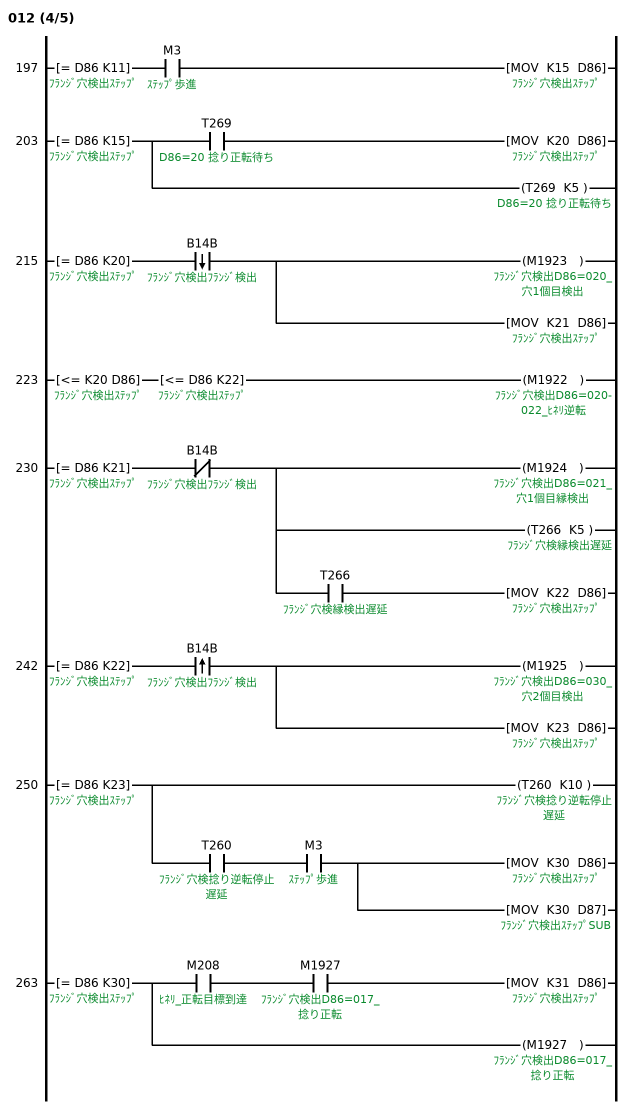
197   LD=     D86 K11  ; ﾌﾗﾝｼﾞ穴検出ｽﾃｯﾌﾟ
      AND     M3  ; ｽﾃｯﾌﾟ歩進
      MOV     K15 D86
203   LD=     D86 K15  ; ﾌﾗﾝｼﾞ穴検出ｽﾃｯﾌﾟ
      MPS
      AND     T269  ; D86=20 捻り正転待ち
      MOV     K20 D86
      MPP
      OUT     T269 K5  ; D86=20 捻り正転待ち
215   LD=     D86 K20  ; ﾌﾗﾝｼﾞ穴検出ｽﾃｯﾌﾟ
      ANDF    B14B  ; ﾌﾗﾝｼﾞ穴検出ﾌﾗﾝｼﾞ検出
      OUT     M1923  ; ﾌﾗﾝｼﾞ穴検出D86=020_穴1個目検出
      MOV     K21 D86
223   LD<=    K20 D86  ; ﾌﾗﾝｼﾞ穴検出ｽﾃｯﾌﾟ
      AND<=   D86 K22  ; ﾌﾗﾝｼﾞ穴検出ｽﾃｯﾌﾟ
      OUT     M1922  ; ﾌﾗﾝｼﾞ穴検出D86=020-022_ﾋﾈﾘ逆転
230   LD=     D86 K21  ; ﾌﾗﾝｼﾞ穴検出ｽﾃｯﾌﾟ
      ANI     B14B  ; ﾌﾗﾝｼﾞ穴検出ﾌﾗﾝｼﾞ検出
      OUT     M1924  ; ﾌﾗﾝｼﾞ穴検出D86=021_穴1個目縁検出
      OUT     T266 K5  ; ﾌﾗﾝｼﾞ穴検縁検出遅延
      AND     T266  ; ﾌﾗﾝｼﾞ穴検縁検出遅延
      MOV     K22 D86
242   LD=     D86 K22  ; ﾌﾗﾝｼﾞ穴検出ｽﾃｯﾌﾟ
      ANDP    B14B  ; ﾌﾗﾝｼﾞ穴検出ﾌﾗﾝｼﾞ検出
      OUT     M1925  ; ﾌﾗﾝｼﾞ穴検出D86=030_穴2個目検出
      MOV     K23 D86
250   LD=     D86 K23  ; ﾌﾗﾝｼﾞ穴検出ｽﾃｯﾌﾟ
      OUT     T260 K10  ; ﾌﾗﾝｼﾞ穴検捻り逆転停止遅延
      AND     T260  ; ﾌﾗﾝｼﾞ穴検捻り逆転停止遅延
      AND     M3  ; ｽﾃｯﾌﾟ歩進
      MOV     K30 D86
      MOV     K30 D87
263   LD=     D86 K30  ; ﾌﾗﾝｼﾞ穴検出ｽﾃｯﾌﾟ
      MPS
      AND     M208  ; ﾋﾈﾘ_正転目標到達
      AND     M1927  ; ﾌﾗﾝｼﾞ穴検出D86=017_捻り正転
      MOV     K31 D86
      MPP
      OUT     M1927  ; ﾌﾗﾝｼﾞ穴検出D86=017_捻り正転
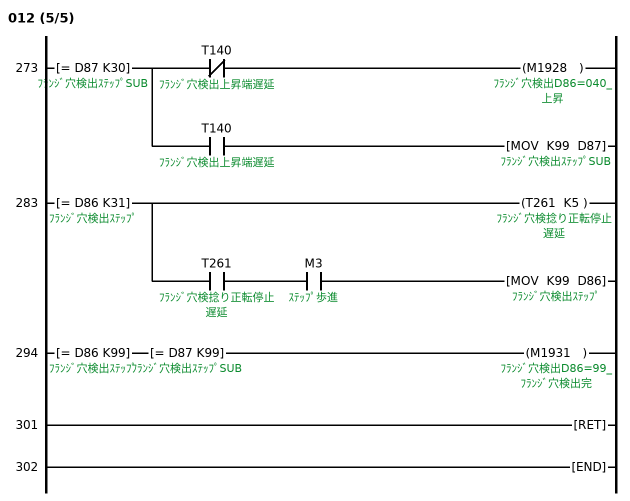
273   LD=     D87 K30  ; ﾌﾗﾝｼﾞ穴検出ｽﾃｯﾌﾟSUB
      MPS
      ANI     T140  ; ﾌﾗﾝｼﾞ穴検出上昇端遅延
      OUT     M1928  ; ﾌﾗﾝｼﾞ穴検出D86=040_上昇
      MPP
      AND     T140  ; ﾌﾗﾝｼﾞ穴検出上昇端遅延
      MOV     K99 D87
283   LD=     D86 K31  ; ﾌﾗﾝｼﾞ穴検出ｽﾃｯﾌﾟ
      OUT     T261 K5  ; ﾌﾗﾝｼﾞ穴検捻り正転停止遅延
      AND     T261  ; ﾌﾗﾝｼﾞ穴検捻り正転停止遅延
      AND     M3  ; ｽﾃｯﾌﾟ歩進
      MOV     K99 D86
294   LD=     D86 K99  ; ﾌﾗﾝｼﾞ穴検出ｽﾃｯﾌﾟ
      AND=    D87 K99  ; ﾌﾗﾝｼﾞ穴検出ｽﾃｯﾌﾟSUB
      OUT     M1931  ; ﾌﾗﾝｼﾞ穴検出D86=99_ﾌﾗﾝｼﾞ穴検出完
301   RET
302   END
END_PROGRAM

PROGRAM 013  // ひねり
; 
      P1300
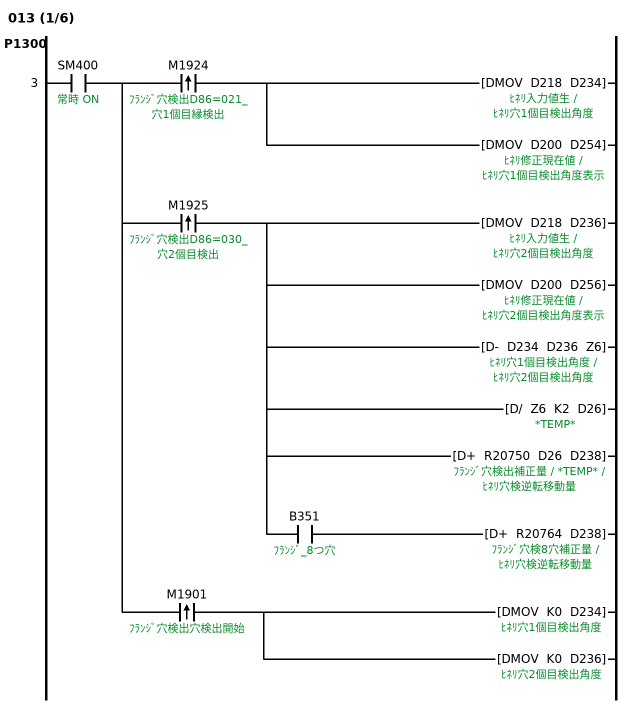
3     LD      SM400  ; 常時 ON
      MPS
      ANDP    M1924  ; ﾌﾗﾝｼﾞ穴検出D86=021_穴1個目縁検出
      DMOV    D218 D234  ; ﾋﾈﾘ入力値生 / ﾋﾈﾘ穴1個目検出角度
      DMOV    D200 D254  ; ﾋﾈﾘ修正現在値 / ﾋﾈﾘ穴1個目検出角度表示
      MRD
      ANDP    M1925  ; ﾌﾗﾝｼﾞ穴検出D86=030_穴2個目検出
      DMOV    D218 D236  ; ﾋﾈﾘ穴2個目検出角度
      DMOV    D200 D256  ; ﾋﾈﾘ穴2個目検出角度表示
      D-      D234 D236 Z6
      D/      Z6 K2 D26  ; *TEMP*
      D+      R20750 D26 D238  ; ﾌﾗﾝｼﾞ穴検出補正量 / ﾋﾈﾘ穴検逆転移動量
      AND     B351  ; ﾌﾗﾝｼﾞ_8つ穴
      D+      R20764 D238  ; ﾌﾗﾝｼﾞ穴検8穴補正量
      MPP
      ANDP    M1901  ; ﾌﾗﾝｼﾞ穴検出穴検出開始
      DMOV    K0 D234
      DMOV    K0 D236
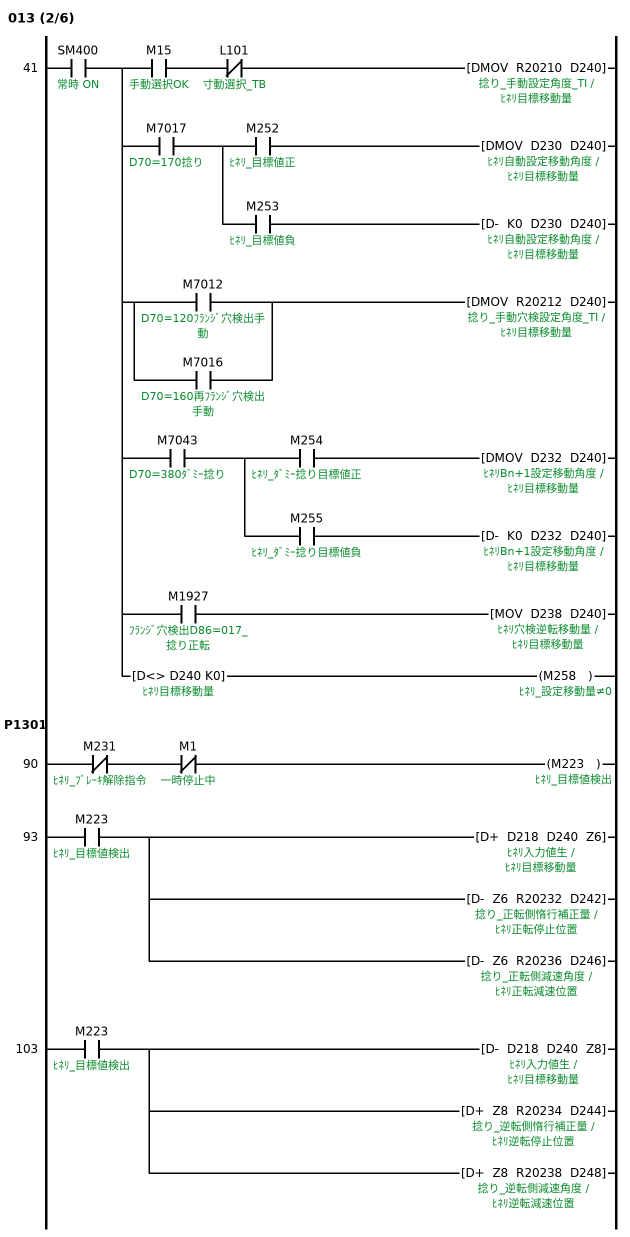
41    LD      SM400  ; 常時 ON
      MPS
      AND     M15  ; 手動選択OK
      ANI     L101  ; 寸動選択_TB
      DMOV    R20210 D240  ; 捻り_手動設定角度_TI / ﾋﾈﾘ目標移動量
      MRD
      AND     M7017  ; D70=170捻り
      MPS
      AND     M252  ; ﾋﾈﾘ_目標値正
      DMOV    D230 D240  ; ﾋﾈﾘ自動設定移動角度
      MPP
      AND     M253  ; ﾋﾈﾘ_目標値負
      D-      K0 D230 D240
      MRD
      LD      M7012  ; D70=120ﾌﾗﾝｼﾞ穴検出手動
      OR      M7016  ; D70=160再ﾌﾗﾝｼﾞ穴検出手動
      ANB
      DMOV    R20212 D240  ; 捻り_手動穴検設定角度_TI
      MRD
      AND     M7043  ; D70=380ﾀﾞﾐｰ捻り
      MPS
      AND     M254  ; ﾋﾈﾘ_ﾀﾞﾐｰ捻り目標値正
      DMOV    D232 D240  ; ﾋﾈﾘBn+1設定移動角度
      MPP
      AND     M255  ; ﾋﾈﾘ_ﾀﾞﾐｰ捻り目標値負
      D-      K0 D232 D240
      MRD
      AND     M1927  ; ﾌﾗﾝｼﾞ穴検出D86=017_捻り正転
      MOV     D238 D240
      MPP
      ANDD<>  D240 K0  ; ﾋﾈﾘ目標移動量
      OUT     M258  ; ﾋﾈﾘ_設定移動量≠0
; 
      P1301
90    LDI     M231  ; ﾋﾈﾘ_ﾌﾞﾚｰｷ解除指令
      ANI     M1  ; 一時停止中
      OUT     M223  ; ﾋﾈﾘ_目標値検出
93    LD      M223  ; ﾋﾈﾘ_目標値検出
      D+      D218 D240 Z6
      D-      Z6 R20232 D242  ; 捻り_正転側惰行補正量 / ﾋﾈﾘ正転停止位置
      D-      Z6 R20236 D246  ; 捻り_正転側減速角度 / ﾋﾈﾘ正転減速位置
103   LD      M223  ; ﾋﾈﾘ_目標値検出
      D-      D218 D240 Z8
      D+      Z8 R20234 D244  ; 捻り_逆転側惰行補正量 / ﾋﾈﾘ逆転停止位置
      D+      Z8 R20238 D248  ; 捻り_逆転側減速角度 / ﾋﾈﾘ逆転減速位置
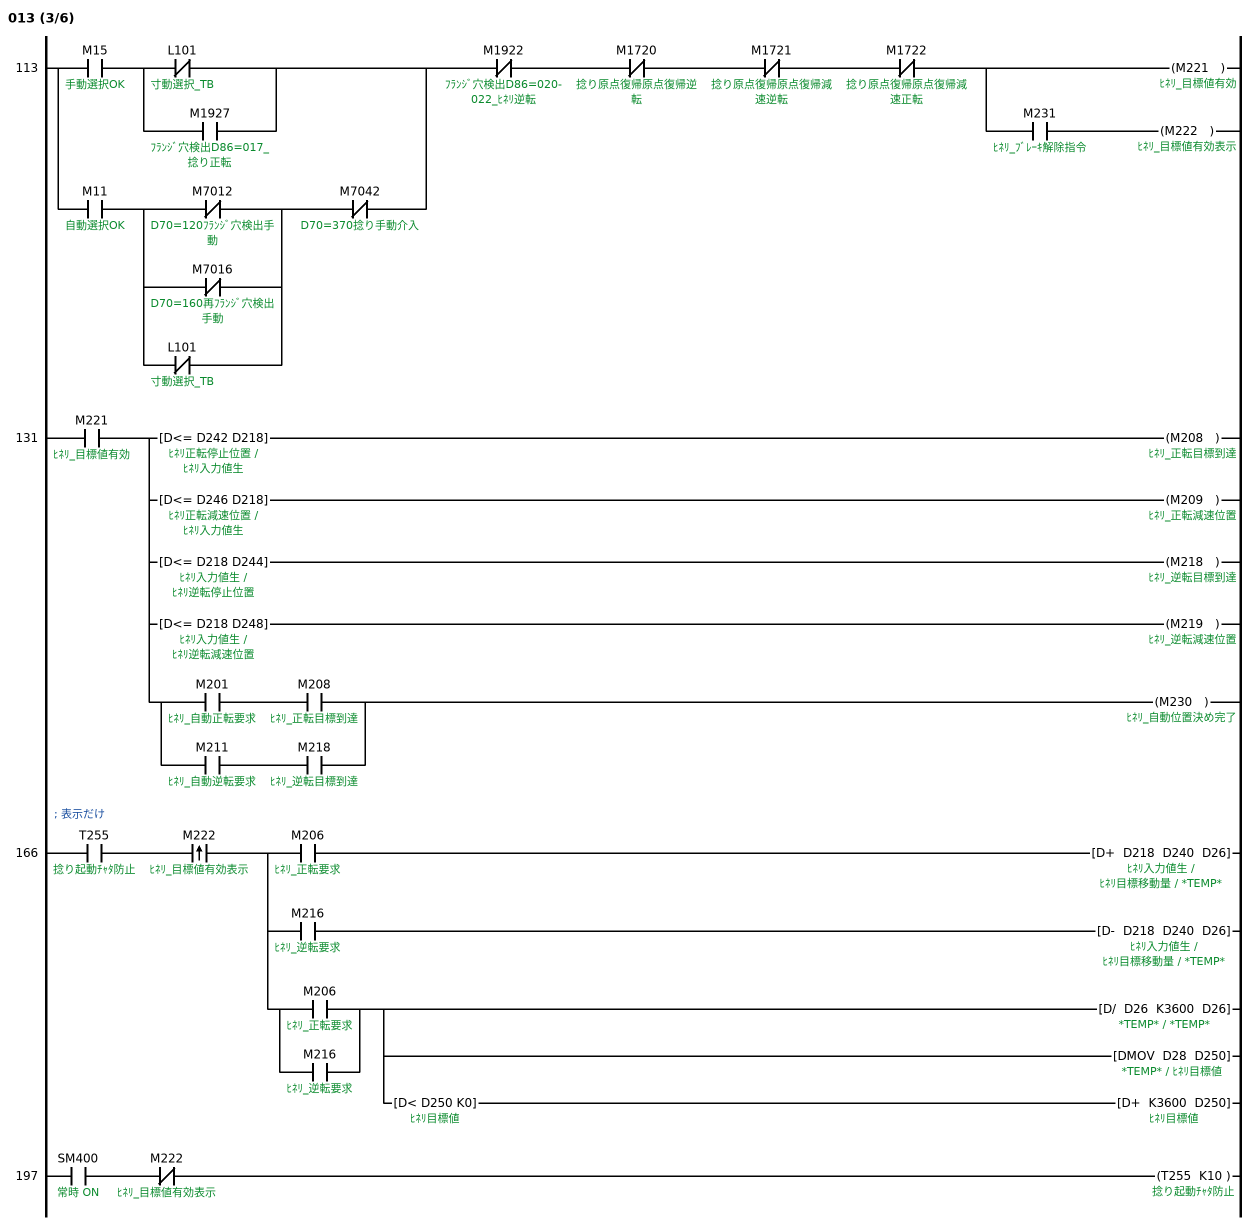
113   LD      M15  ; 手動選択OK
      LDI     L101  ; 寸動選択_TB
      OR      M1927  ; ﾌﾗﾝｼﾞ穴検出D86=017_捻り正転
      ANB
      LD      M11  ; 自動選択OK
      LDI     M7012  ; D70=120ﾌﾗﾝｼﾞ穴検出手動
      ORI     M7016  ; D70=160再ﾌﾗﾝｼﾞ穴検出手動
      ORI     L101  ; 寸動選択_TB
      ANB
      ANI     M7042  ; D70=370捻り手動介入
      ORB
      ANI     M1922  ; ﾌﾗﾝｼﾞ穴検出D86=020-022_ﾋﾈﾘ逆転
      ANI     M1720  ; 捻り原点復帰原点復帰逆転
      ANI     M1721  ; 捻り原点復帰原点復帰減速逆転
      ANI     M1722  ; 捻り原点復帰原点復帰減速正転
      OUT     M221  ; ﾋﾈﾘ_目標値有効
      AND     M231  ; ﾋﾈﾘ_ﾌﾞﾚｰｷ解除指令
      OUT     M222  ; ﾋﾈﾘ_目標値有効表示
131   LD      M221  ; ﾋﾈﾘ_目標値有効
      MPS
      ANDD<=  D242 D218  ; ﾋﾈﾘ正転停止位置 / ﾋﾈﾘ入力値生
      OUT     M208  ; ﾋﾈﾘ_正転目標到達
      MRD
      ANDD<=  D246 D218  ; ﾋﾈﾘ正転減速位置 / ﾋﾈﾘ入力値生
      OUT     M209  ; ﾋﾈﾘ_正転減速位置
      MRD
      ANDD<=  D218 D244  ; ﾋﾈﾘ入力値生 / ﾋﾈﾘ逆転停止位置
      OUT     M218  ; ﾋﾈﾘ_逆転目標到達
      MRD
      ANDD<=  D218 D248  ; ﾋﾈﾘ入力値生 / ﾋﾈﾘ逆転減速位置
      OUT     M219  ; ﾋﾈﾘ_逆転減速位置
      MPP
      LD      M201  ; ﾋﾈﾘ_自動正転要求
      AND     M208  ; ﾋﾈﾘ_正転目標到達
      LD      M211  ; ﾋﾈﾘ_自動逆転要求
      AND     M218  ; ﾋﾈﾘ_逆転目標到達
      ORB
      ANB
      OUT     M230  ; ﾋﾈﾘ_自動位置決め完了
; 表示だけ
166   LD      T255  ; 捻り起動ﾁｬﾀ防止
      ANDP    M222  ; ﾋﾈﾘ_目標値有効表示
      MPS
      AND     M206  ; ﾋﾈﾘ_正転要求
      D+      D218 D240 D26
      MRD
      AND     M216  ; ﾋﾈﾘ_逆転要求
      D-      D218 D240 D26
      MPP
      LD      M206  ; ﾋﾈﾘ_正転要求
      OR      M216  ; ﾋﾈﾘ_逆転要求
      ANB
      D/      D26 K3600 D26
      DMOV    D28 D250  ; *TEMP* / ﾋﾈﾘ目標値
      ANDD<   D250 K0  ; ﾋﾈﾘ目標値
      D+      K3600 D250
197   LD      SM400  ; 常時 ON
      ANI     M222  ; ﾋﾈﾘ_目標値有効表示
      OUT     T255 K10  ; 捻り起動ﾁｬﾀ防止
; 
      P1302
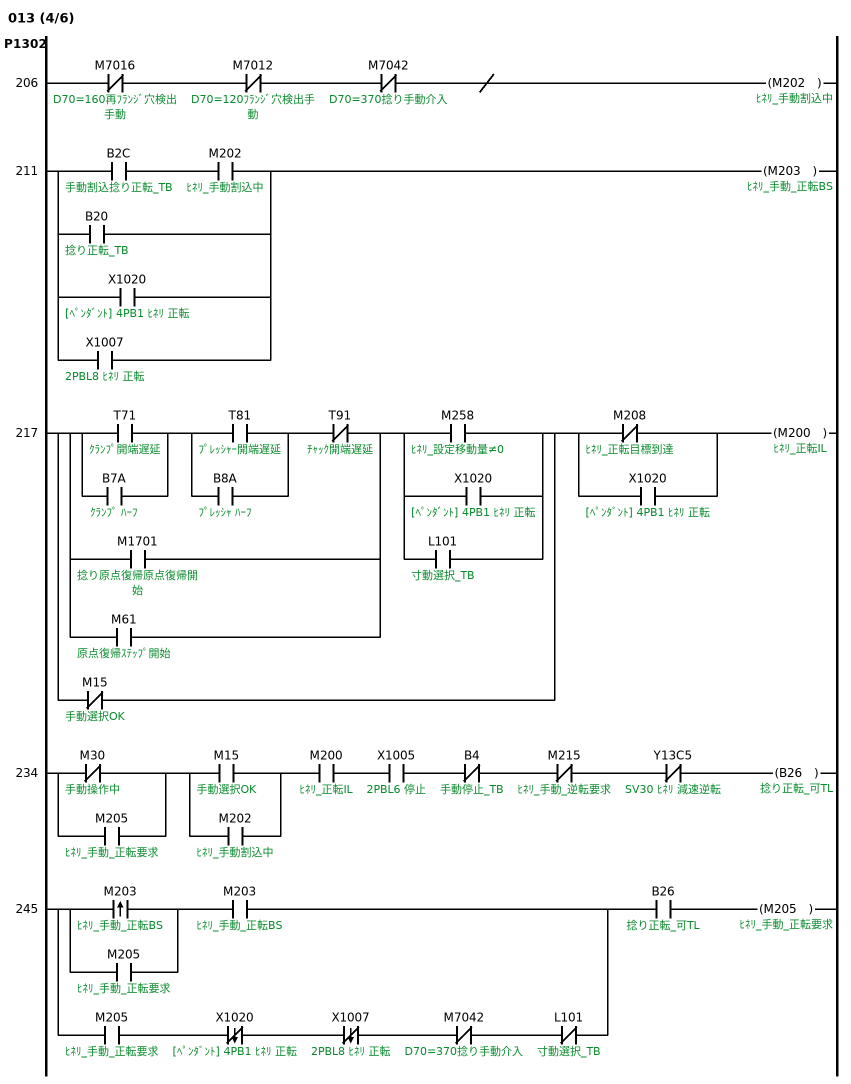
206   LDI     M7016  ; D70=160再ﾌﾗﾝｼﾞ穴検出手動
      ANI     M7012  ; D70=120ﾌﾗﾝｼﾞ穴検出手動
      ANI     M7042  ; D70=370捻り手動介入
      INV
      OUT     M202  ; ﾋﾈﾘ_手動割込中
211   LD      B2C  ; 手動割込捻り正転_TB
      AND     M202  ; ﾋﾈﾘ_手動割込中
      OR      B20  ; 捻り正転_TB
      OR      X1020  ; [ﾍﾟﾝﾀﾞﾝﾄ] 4PB1 ﾋﾈﾘ 正転
      OR      X1007  ; 2PBL8 ﾋﾈﾘ 正転
      OUT     M203  ; ﾋﾈﾘ_手動_正転BS
217   LD      T71  ; ｸﾗﾝﾌﾟ開端遅延
      OR      B7A  ; ｸﾗﾝﾌﾟ ﾊｰﾌ
      LD      T81  ; ﾌﾟﾚｯｼｬｰ開端遅延
      OR      B8A  ; ﾌﾟﾚｯｼｬ ﾊｰﾌ
      ANB
      ANI     T91  ; ﾁｬｯｸ開端遅延
      OR      M1701  ; 捻り原点復帰原点復帰開始
      OR      M61  ; 原点復帰ｽﾃｯﾌﾟ開始
      LD      M258  ; ﾋﾈﾘ_設定移動量≠0
      OR      X1020  ; [ﾍﾟﾝﾀﾞﾝﾄ] 4PB1 ﾋﾈﾘ 正転
      OR      L101  ; 寸動選択_TB
      ANB
      ORI     M15  ; 手動選択OK
      LDI     M208  ; ﾋﾈﾘ_正転目標到達
      OR      X1020  ; [ﾍﾟﾝﾀﾞﾝﾄ] 4PB1 ﾋﾈﾘ 正転
      ANB
      OUT     M200  ; ﾋﾈﾘ_正転IL
234   LDI     M30  ; 手動操作中
      OR      M205  ; ﾋﾈﾘ_手動_正転要求
      LD      M15  ; 手動選択OK
      OR      M202  ; ﾋﾈﾘ_手動割込中
      ANB
      AND     M200  ; ﾋﾈﾘ_正転IL
      AND     X1005  ; 2PBL6 停止
      ANI     B4  ; 手動停止_TB
      ANI     M215  ; ﾋﾈﾘ_手動_逆転要求
      ANI     Y13C5  ; SV30 ﾋﾈﾘ 減速逆転
      OUT     B26  ; 捻り正転_可TL
245   LDP     M203  ; ﾋﾈﾘ_手動_正転BS
      OR      M205  ; ﾋﾈﾘ_手動_正転要求
      AND     M203  ; ﾋﾈﾘ_手動_正転BS
      LD      M205  ; ﾋﾈﾘ_手動_正転要求
      ANDFI   X1020  ; [ﾍﾟﾝﾀﾞﾝﾄ] 4PB1 ﾋﾈﾘ 正転
      ANDFI   X1007  ; 2PBL8 ﾋﾈﾘ 正転
      ANI     M7042  ; D70=370捻り手動介入
      ANI     L101  ; 寸動選択_TB
      ORB
      AND     B26  ; 捻り正転_可TL
      OUT     M205  ; ﾋﾈﾘ_手動_正転要求
; 
      P1303
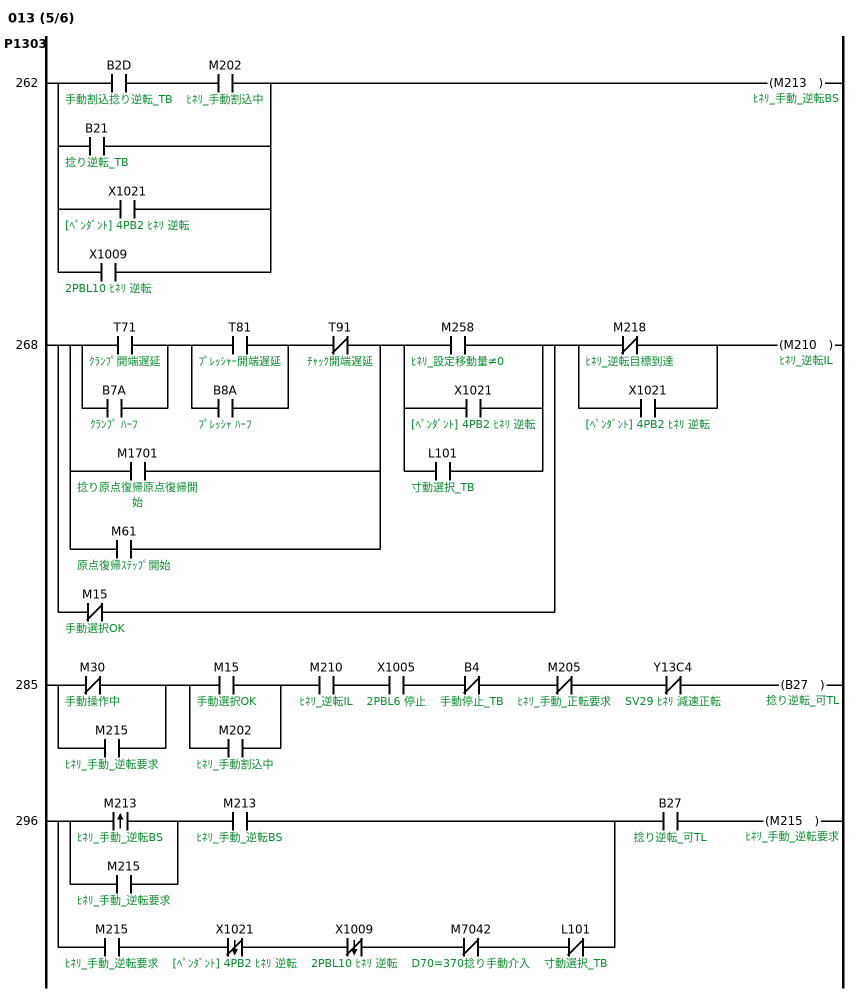
262   LD      B2D  ; 手動割込捻り逆転_TB
      AND     M202  ; ﾋﾈﾘ_手動割込中
      OR      B21  ; 捻り逆転_TB
      OR      X1021  ; [ﾍﾟﾝﾀﾞﾝﾄ] 4PB2 ﾋﾈﾘ 逆転
      OR      X1009  ; 2PBL10 ﾋﾈﾘ 逆転
      OUT     M213  ; ﾋﾈﾘ_手動_逆転BS
268   LD      T71  ; ｸﾗﾝﾌﾟ開端遅延
      OR      B7A  ; ｸﾗﾝﾌﾟ ﾊｰﾌ
      LD      T81  ; ﾌﾟﾚｯｼｬｰ開端遅延
      OR      B8A  ; ﾌﾟﾚｯｼｬ ﾊｰﾌ
      ANB
      ANI     T91  ; ﾁｬｯｸ開端遅延
      OR      M1701  ; 捻り原点復帰原点復帰開始
      OR      M61  ; 原点復帰ｽﾃｯﾌﾟ開始
      LD      M258  ; ﾋﾈﾘ_設定移動量≠0
      OR      X1021  ; [ﾍﾟﾝﾀﾞﾝﾄ] 4PB2 ﾋﾈﾘ 逆転
      OR      L101  ; 寸動選択_TB
      ANB
      ORI     M15  ; 手動選択OK
      LDI     M218  ; ﾋﾈﾘ_逆転目標到達
      OR      X1021  ; [ﾍﾟﾝﾀﾞﾝﾄ] 4PB2 ﾋﾈﾘ 逆転
      ANB
      OUT     M210  ; ﾋﾈﾘ_逆転IL
285   LDI     M30  ; 手動操作中
      OR      M215  ; ﾋﾈﾘ_手動_逆転要求
      LD      M15  ; 手動選択OK
      OR      M202  ; ﾋﾈﾘ_手動割込中
      ANB
      AND     M210  ; ﾋﾈﾘ_逆転IL
      AND     X1005  ; 2PBL6 停止
      ANI     B4  ; 手動停止_TB
      ANI     M205  ; ﾋﾈﾘ_手動_正転要求
      ANI     Y13C4  ; SV29 ﾋﾈﾘ 減速正転
      OUT     B27  ; 捻り逆転_可TL
296   LDP     M213  ; ﾋﾈﾘ_手動_逆転BS
      OR      M215  ; ﾋﾈﾘ_手動_逆転要求
      AND     M213  ; ﾋﾈﾘ_手動_逆転BS
      LD      M215  ; ﾋﾈﾘ_手動_逆転要求
      ANDFI   X1021  ; [ﾍﾟﾝﾀﾞﾝﾄ] 4PB2 ﾋﾈﾘ 逆転
      ANDFI   X1009  ; 2PBL10 ﾋﾈﾘ 逆転
      ANI     M7042  ; D70=370捻り手動介入
      ANI     L101  ; 寸動選択_TB
      ORB
      AND     B27  ; 捻り逆転_可TL
      OUT     M215  ; ﾋﾈﾘ_手動_逆転要求
; 
      P1306
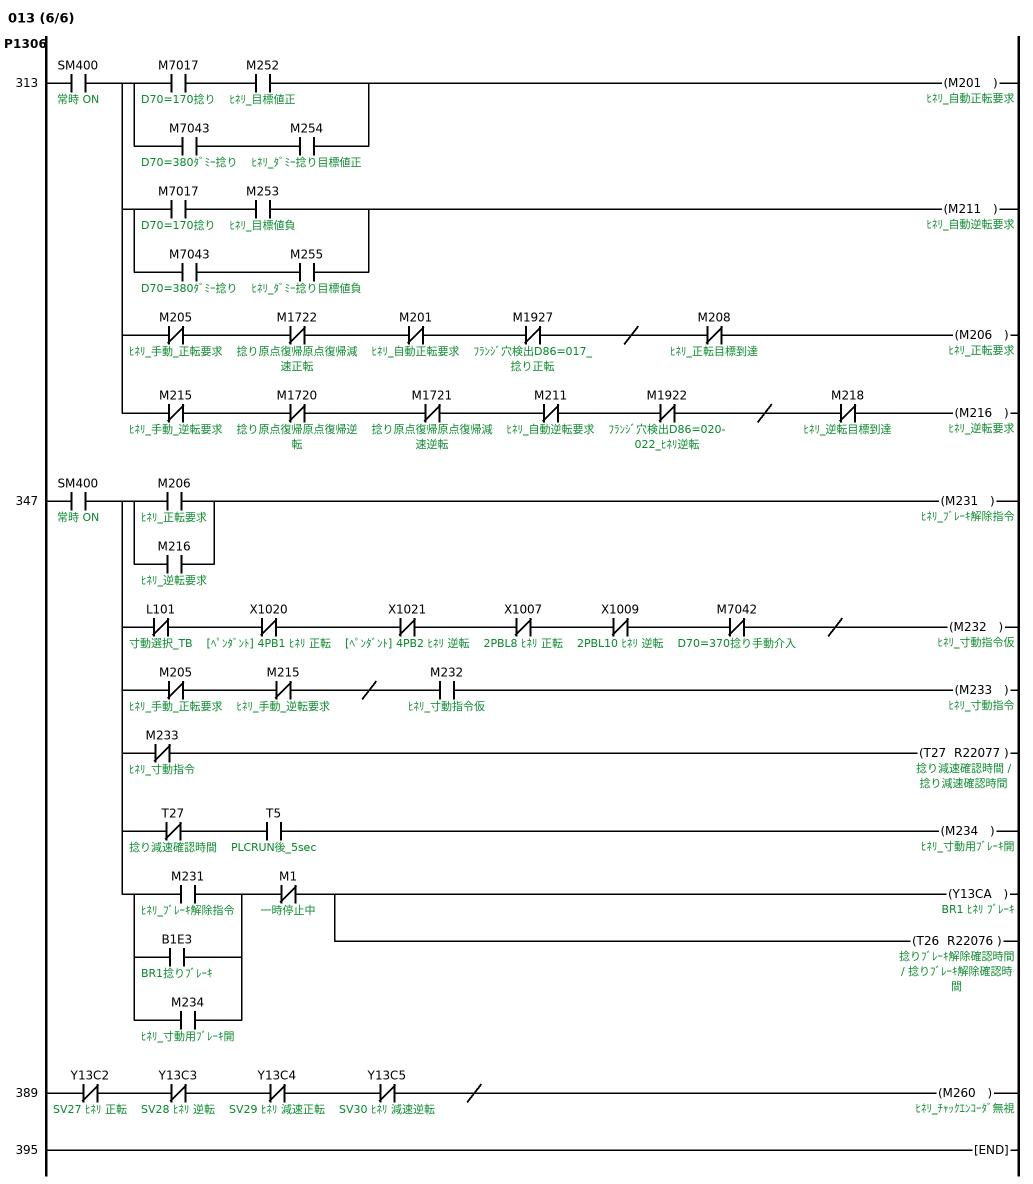
313   LD      SM400  ; 常時 ON
      MPS
      LD      M7017  ; D70=170捻り
      AND     M252  ; ﾋﾈﾘ_目標値正
      LD      M7043  ; D70=380ﾀﾞﾐｰ捻り
      AND     M254  ; ﾋﾈﾘ_ﾀﾞﾐｰ捻り目標値正
      ORB
      ANB
      OUT     M201  ; ﾋﾈﾘ_自動正転要求
      MRD
      LD      M7017  ; D70=170捻り
      AND     M253  ; ﾋﾈﾘ_目標値負
      LD      M7043  ; D70=380ﾀﾞﾐｰ捻り
      AND     M255  ; ﾋﾈﾘ_ﾀﾞﾐｰ捻り目標値負
      ORB
      ANB
      OUT     M211  ; ﾋﾈﾘ_自動逆転要求
      MRD
      ANI     M205  ; ﾋﾈﾘ_手動_正転要求
      ANI     M1722  ; 捻り原点復帰原点復帰減速正転
      ANI     M201  ; ﾋﾈﾘ_自動正転要求
      ANI     M1927  ; ﾌﾗﾝｼﾞ穴検出D86=017_捻り正転
      INV
      ANI     M208  ; ﾋﾈﾘ_正転目標到達
      OUT     M206  ; ﾋﾈﾘ_正転要求
      MPP
      ANI     M215  ; ﾋﾈﾘ_手動_逆転要求
      ANI     M1720  ; 捻り原点復帰原点復帰逆転
      ANI     M1721  ; 捻り原点復帰原点復帰減速逆転
      ANI     M211  ; ﾋﾈﾘ_自動逆転要求
      ANI     M1922  ; ﾌﾗﾝｼﾞ穴検出D86=020-022_ﾋﾈﾘ逆転
      INV
      ANI     M218  ; ﾋﾈﾘ_逆転目標到達
      OUT     M216  ; ﾋﾈﾘ_逆転要求
347   LD      SM400  ; 常時 ON
      MPS
      LD      M206  ; ﾋﾈﾘ_正転要求
      OR      M216  ; ﾋﾈﾘ_逆転要求
      ANB
      OUT     M231  ; ﾋﾈﾘ_ﾌﾞﾚｰｷ解除指令
      MRD
      ANI     L101  ; 寸動選択_TB
      ANI     X1020  ; [ﾍﾟﾝﾀﾞﾝﾄ] 4PB1 ﾋﾈﾘ 正転
      ANI     X1021  ; [ﾍﾟﾝﾀﾞﾝﾄ] 4PB2 ﾋﾈﾘ 逆転
      ANI     X1007  ; 2PBL8 ﾋﾈﾘ 正転
      ANI     X1009  ; 2PBL10 ﾋﾈﾘ 逆転
      ANI     M7042  ; D70=370捻り手動介入
      INV
      OUT     M232  ; ﾋﾈﾘ_寸動指令仮
      MRD
      ANI     M205  ; ﾋﾈﾘ_手動_正転要求
      ANI     M215  ; ﾋﾈﾘ_手動_逆転要求
      INV
      AND     M232  ; ﾋﾈﾘ_寸動指令仮
      OUT     M233  ; ﾋﾈﾘ_寸動指令
      MRD
      ANI     M233  ; ﾋﾈﾘ_寸動指令
      OUT     T27 R22077  ; 捻り減速確認時間 / 捻り減速確認時間
      MRD
      ANI     T27  ; 捻り減速確認時間
      AND     T5  ; PLCRUN後_5sec
      OUT     M234  ; ﾋﾈﾘ_寸動用ﾌﾞﾚｰｷ開
      MPP
      LD      M231  ; ﾋﾈﾘ_ﾌﾞﾚｰｷ解除指令
      OR      B1E3  ; BR1捻りﾌﾞﾚｰｷ
      OR      M234  ; ﾋﾈﾘ_寸動用ﾌﾞﾚｰｷ開
      ANB
      ANI     M1  ; 一時停止中
      OUT     Y13CA  ; BR1 ﾋﾈﾘ ﾌﾞﾚｰｷ
      OUT     T26 R22076  ; 捻りﾌﾞﾚｰｷ解除確認時間 / 捻りﾌﾞﾚｰｷ解除確認時間
389   LDI     Y13C2  ; SV27 ﾋﾈﾘ 正転
      ANI     Y13C3  ; SV28 ﾋﾈﾘ 逆転
      ANI     Y13C4  ; SV29 ﾋﾈﾘ 減速正転
      ANI     Y13C5  ; SV30 ﾋﾈﾘ 減速逆転
      INV
      OUT     M260  ; ﾋﾈﾘ_ﾁｬｯｸｴﾝｺｰﾀﾞ無視
395   END
END_PROGRAM

PROGRAM 018  // 送り
; 
      P1802
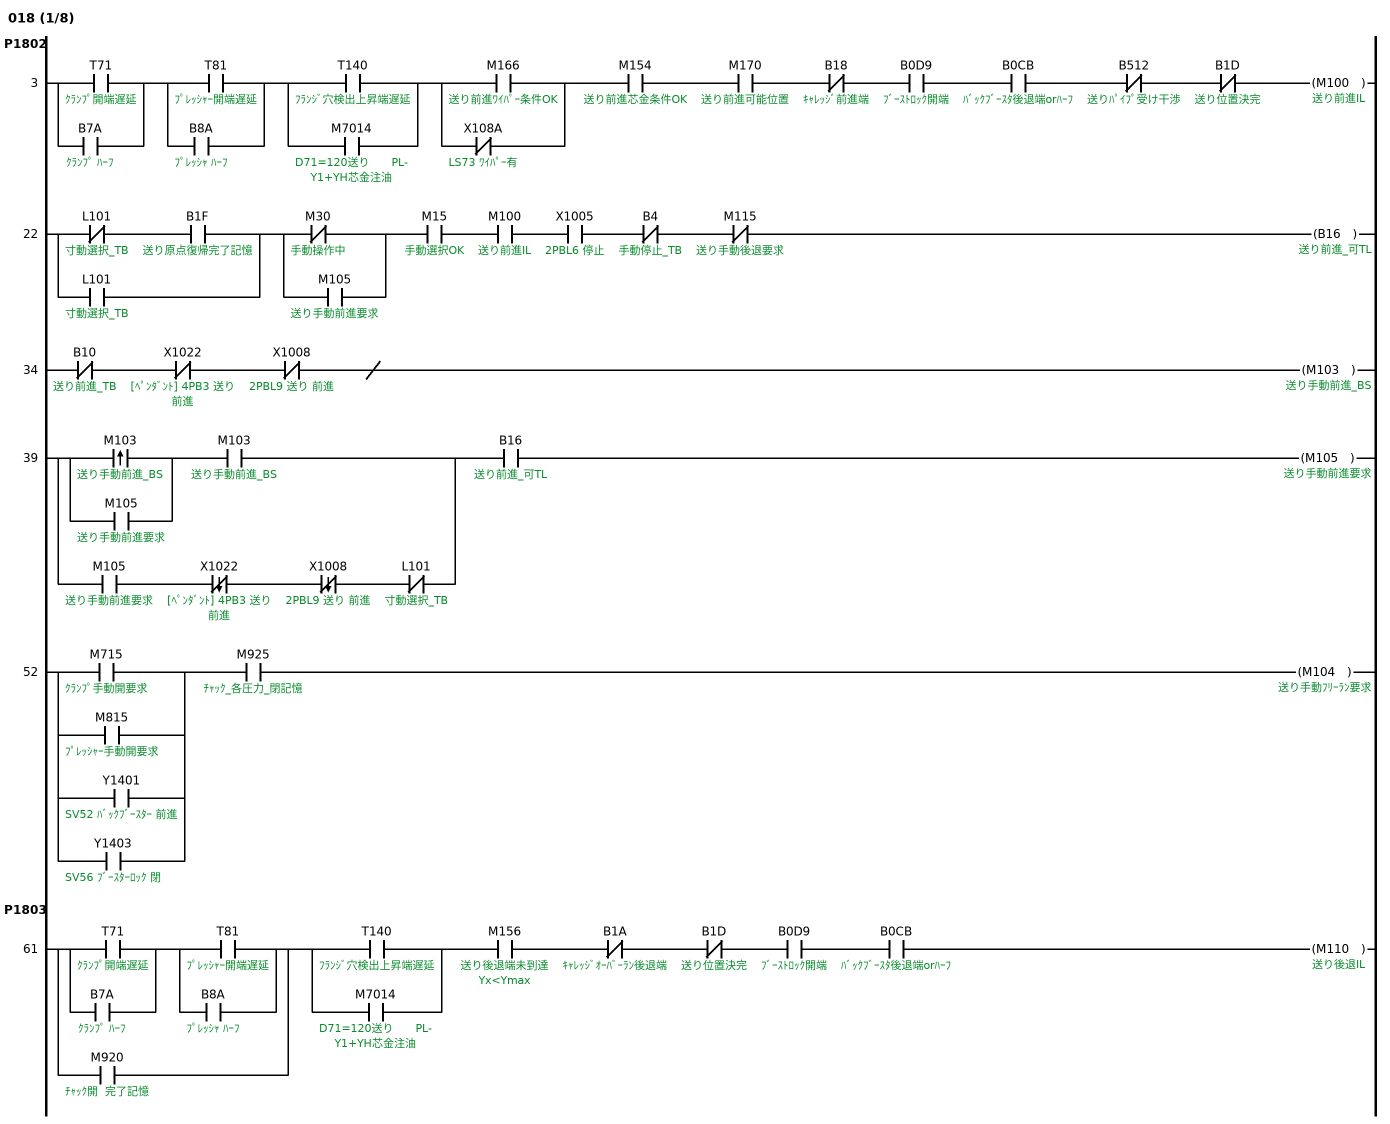
3     LD      T71  ; ｸﾗﾝﾌﾟ開端遅延
      OR      B7A  ; ｸﾗﾝﾌﾟ ﾊｰﾌ
      LD      T81  ; ﾌﾟﾚｯｼｬｰ開端遅延
      OR      B8A  ; ﾌﾟﾚｯｼｬ ﾊｰﾌ
      ANB
      LD      T140  ; ﾌﾗﾝｼﾞ穴検出上昇端遅延
      OR      M7014  ; D71=120送り　　PL-Y1+YH芯金注油
      ANB
      LD      M166  ; 送り前進ﾜｲﾊﾟｰ条件OK
      ORI     X108A  ; LS73 ﾜｲﾊﾟｰ有
      ANB
      AND     M154  ; 送り前進芯金条件OK
      AND     M170  ; 送り前進可能位置
      ANI     B18  ; ｷｬﾚｯｼﾞ前進端
      AND     B0D9  ; ﾌﾞｰｽﾄﾛｯｸ開端
      AND     B0CB  ; ﾊﾞｯｸﾌﾞｰｽﾀ後退端orﾊｰﾌ
      ANI     B512  ; 送りﾊﾟｲﾌﾟ受け干渉
      ANI     B1D  ; 送り位置決完
      OUT     M100  ; 送り前進IL
22    LDI     L101  ; 寸動選択_TB
      AND     B1F  ; 送り原点復帰完了記憶
      OR      L101  ; 寸動選択_TB
      LDI     M30  ; 手動操作中
      OR      M105  ; 送り手動前進要求
      ANB
      AND     M15  ; 手動選択OK
      AND     M100  ; 送り前進IL
      AND     X1005  ; 2PBL6 停止
      ANI     B4  ; 手動停止_TB
      ANI     M115  ; 送り手動後退要求
      OUT     B16  ; 送り前進_可TL
34    LDI     B10  ; 送り前進_TB
      ANI     X1022  ; [ﾍﾟﾝﾀﾞﾝﾄ] 4PB3 送り 前進
      ANI     X1008  ; 2PBL9 送り 前進
      INV
      OUT     M103  ; 送り手動前進_BS
39    LDP     M103  ; 送り手動前進_BS
      OR      M105  ; 送り手動前進要求
      AND     M103  ; 送り手動前進_BS
      LD      M105  ; 送り手動前進要求
      ANDFI   X1022  ; [ﾍﾟﾝﾀﾞﾝﾄ] 4PB3 送り 前進
      ANDFI   X1008  ; 2PBL9 送り 前進
      ANI     L101  ; 寸動選択_TB
      ORB
      AND     B16  ; 送り前進_可TL
      OUT     M105  ; 送り手動前進要求
52    LD      M715  ; ｸﾗﾝﾌﾟ手動開要求
      OR      M815  ; ﾌﾟﾚｯｼｬｰ手動開要求
      OR      Y1401  ; SV52 ﾊﾞｯｸﾌﾞｰｽﾀｰ 前進
      OR      Y1403  ; SV56 ﾌﾞｰｽﾀｰﾛｯｸ 閉
      AND     M925  ; ﾁｬｯｸ_各圧力_閉記憶
      OUT     M104  ; 送り手動ﾌﾘｰﾗﾝ要求
; 
      P1803
61    LD      T71  ; ｸﾗﾝﾌﾟ開端遅延
      OR      B7A  ; ｸﾗﾝﾌﾟ ﾊｰﾌ
      LD      T81  ; ﾌﾟﾚｯｼｬｰ開端遅延
      OR      B8A  ; ﾌﾟﾚｯｼｬ ﾊｰﾌ
      ANB
      OR      M920  ; ﾁｬｯｸ開  完了記憶
      LD      T140  ; ﾌﾗﾝｼﾞ穴検出上昇端遅延
      OR      M7014  ; D71=120送り　　PL-Y1+YH芯金注油
      ANB
      AND     M156  ; 送り後退端未到達 Yx<Ymax
      ANI     B1A  ; ｷｬﾚｯｼﾞｵｰﾊﾞｰﾗﾝ後退端
      ANI     B1D  ; 送り位置決完
      AND     B0D9  ; ﾌﾞｰｽﾄﾛｯｸ開端
      AND     B0CB  ; ﾊﾞｯｸﾌﾞｰｽﾀ後退端orﾊｰﾌ
      OUT     M110  ; 送り後退IL
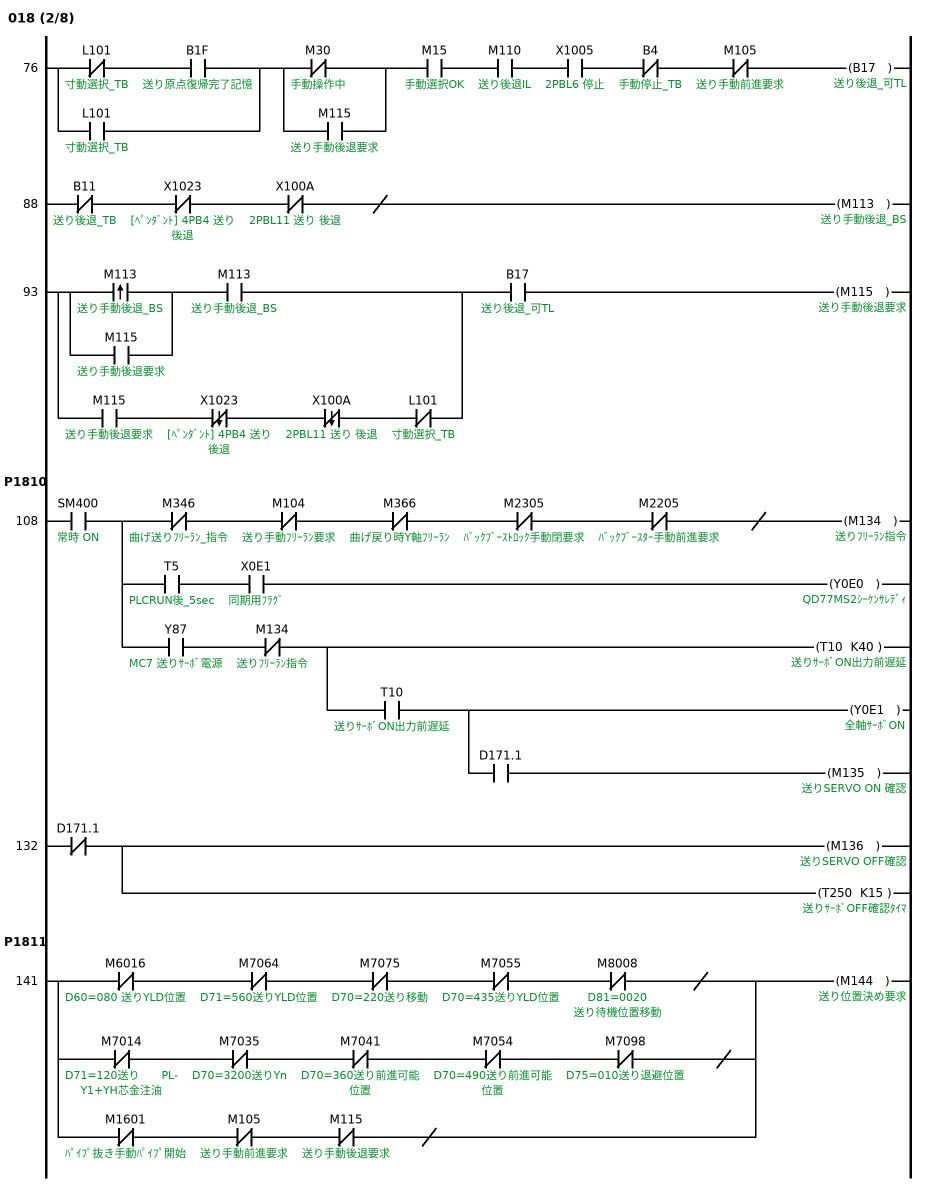
76    LDI     L101  ; 寸動選択_TB
      AND     B1F  ; 送り原点復帰完了記憶
      OR      L101  ; 寸動選択_TB
      LDI     M30  ; 手動操作中
      OR      M115  ; 送り手動後退要求
      ANB
      AND     M15  ; 手動選択OK
      AND     M110  ; 送り後退IL
      AND     X1005  ; 2PBL6 停止
      ANI     B4  ; 手動停止_TB
      ANI     M105  ; 送り手動前進要求
      OUT     B17  ; 送り後退_可TL
88    LDI     B11  ; 送り後退_TB
      ANI     X1023  ; [ﾍﾟﾝﾀﾞﾝﾄ] 4PB4 送り 後退
      ANI     X100A  ; 2PBL11 送り 後退
      INV
      OUT     M113  ; 送り手動後退_BS
93    LDP     M113  ; 送り手動後退_BS
      OR      M115  ; 送り手動後退要求
      AND     M113  ; 送り手動後退_BS
      LD      M115  ; 送り手動後退要求
      ANDFI   X1023  ; [ﾍﾟﾝﾀﾞﾝﾄ] 4PB4 送り 後退
      ANDFI   X100A  ; 2PBL11 送り 後退
      ANI     L101  ; 寸動選択_TB
      ORB
      AND     B17  ; 送り後退_可TL
      OUT     M115  ; 送り手動後退要求
; 
      P1810
108   LD      SM400  ; 常時 ON
      MPS
      ANI     M346  ; 曲げ送りﾌﾘｰﾗﾝ_指令
      ANI     M104  ; 送り手動ﾌﾘｰﾗﾝ要求
      ANI     M366  ; 曲げ戻り時Y軸ﾌﾘｰﾗﾝ
      ANI     M2305  ; ﾊﾞｯｸﾌﾞｰｽﾄﾛｯｸ手動閉要求
      ANI     M2205  ; ﾊﾞｯｸﾌﾞｰｽﾀｰ手動前進要求
      INV
      OUT     M134  ; 送りﾌﾘｰﾗﾝ指令
      MRD
      AND     T5  ; PLCRUN後_5sec
      AND     X0E1  ; 同期用ﾌﾗｸﾞ
      OUT     Y0E0  ; QD77MS2ｼｰｹﾝｻﾚﾃﾞｨ
      MPP
      AND     Y87  ; MC7 送りｻｰﾎﾞ電源
      ANI     M134  ; 送りﾌﾘｰﾗﾝ指令
      OUT     T10 K40  ; 送りｻｰﾎﾞON出力前遅延
      AND     T10  ; 送りｻｰﾎﾞON出力前遅延
      OUT     Y0E1  ; 全軸ｻｰﾎﾞON
      AND     D171.1
      OUT     M135  ; 送りSERVO ON 確認
132   LDI     D171.1
      OUT     M136  ; 送りSERVO OFF確認
      OUT     T250 K15  ; 送りｻｰﾎﾞOFF確認ﾀｲﾏ
; 
      P1811
141   LDI     M6016  ; D60=080 送りYLD位置
      ANI     M7064  ; D71=560送りYLD位置
      ANI     M7075  ; D70=220送り移動
      ANI     M7055  ; D70=435送りYLD位置
      ANI     M8008  ; D81=0020 送り待機位置移動
      INV
      LDI     M7014  ; D71=120送り　　PL-Y1+YH芯金注油
      ANI     M7035  ; D70=3200送りYn
      ANI     M7041  ; D70=360送り前進可能位置
      ANI     M7054  ; D70=490送り前進可能位置
      ANI     M7098  ; D75=010送り退避位置
      INV
      ORB
      LDI     M1601  ; ﾊﾟｲﾌﾟ抜き手動ﾊﾟｲﾌﾟ開始
      ANI     M105  ; 送り手動前進要求
      ANI     M115  ; 送り手動後退要求
      INV
      ORB
      OUT     M144  ; 送り位置決め要求
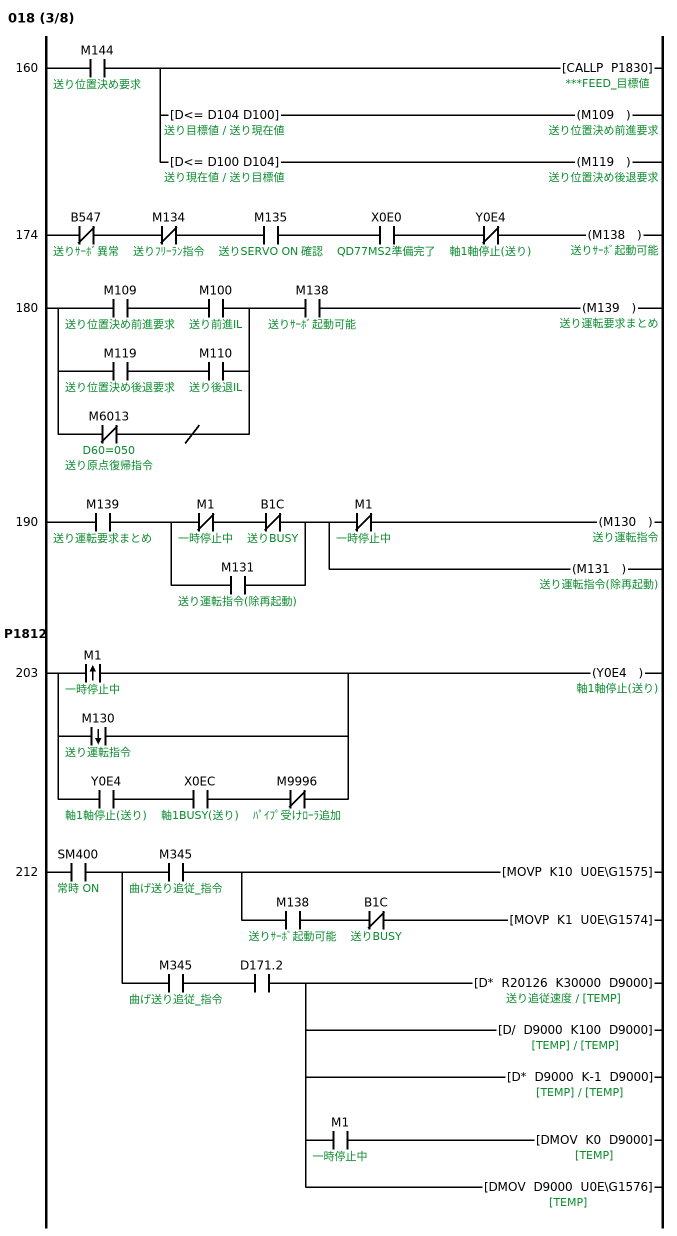
160   LD      M144  ; 送り位置決め要求
      CALLP   P1830  ; ***FEED_目標値
      MPS
      ANDD<=  D104 D100  ; 送り目標値 / 送り現在値
      OUT     M109  ; 送り位置決め前進要求
      MPP
      ANDD<=  D100 D104  ; 送り現在値 / 送り目標値
      OUT     M119  ; 送り位置決め後退要求
174   LDI     B547  ; 送りｻｰﾎﾞ異常
      ANI     M134  ; 送りﾌﾘｰﾗﾝ指令
      AND     M135  ; 送りSERVO ON 確認
      AND     X0E0  ; QD77MS2準備完了
      ANI     Y0E4  ; 軸1軸停止(送り)
      OUT     M138  ; 送りｻｰﾎﾞ起動可能
180   LD      M109  ; 送り位置決め前進要求
      AND     M100  ; 送り前進IL
      LD      M119  ; 送り位置決め後退要求
      AND     M110  ; 送り後退IL
      ORB
      LDI     M6013  ; D60=050 送り原点復帰指令
      INV
      ORB
      AND     M138  ; 送りｻｰﾎﾞ起動可能
      OUT     M139  ; 送り運転要求まとめ
190   LD      M139  ; 送り運転要求まとめ
      LDI     M1  ; 一時停止中
      ANI     B1C  ; 送りBUSY
      OR      M131  ; 送り運転指令(除再起動)
      ANB
      MPS
      ANI     M1  ; 一時停止中
      OUT     M130  ; 送り運転指令
      MPP
      OUT     M131  ; 送り運転指令(除再起動)
; 
      P1812
203   LDP     M1  ; 一時停止中
      ORF     M130  ; 送り運転指令
      LD      Y0E4  ; 軸1軸停止(送り)
      AND     X0EC  ; 軸1BUSY(送り)
      ANI     M9996  ; ﾊﾟｲﾌﾟ受けﾛｰﾗ追加
      ORB
      OUT     Y0E4  ; 軸1軸停止(送り)
212   LD      SM400  ; 常時 ON
      MPS
      AND     M345  ; 曲げ送り追従_指令
      MOVP    K10 U0E\G1575
      AND     M138  ; 送りｻｰﾎﾞ起動可能
      ANI     B1C  ; 送りBUSY
      MOVP    K1 U0E\G1574
      MPP
      AND     M345  ; 曲げ送り追従_指令
      AND     D171.2
      D*      R20126 K30000 D9000  ; 送り追従速度 / [TEMP]
      D/      D9000 K100 D9000
      D*      D9000 K-1 D9000
      MPS
      AND     M1  ; 一時停止中
      DMOV    K0 D9000
      MPP
      DMOV    D9000 U0E\G1576
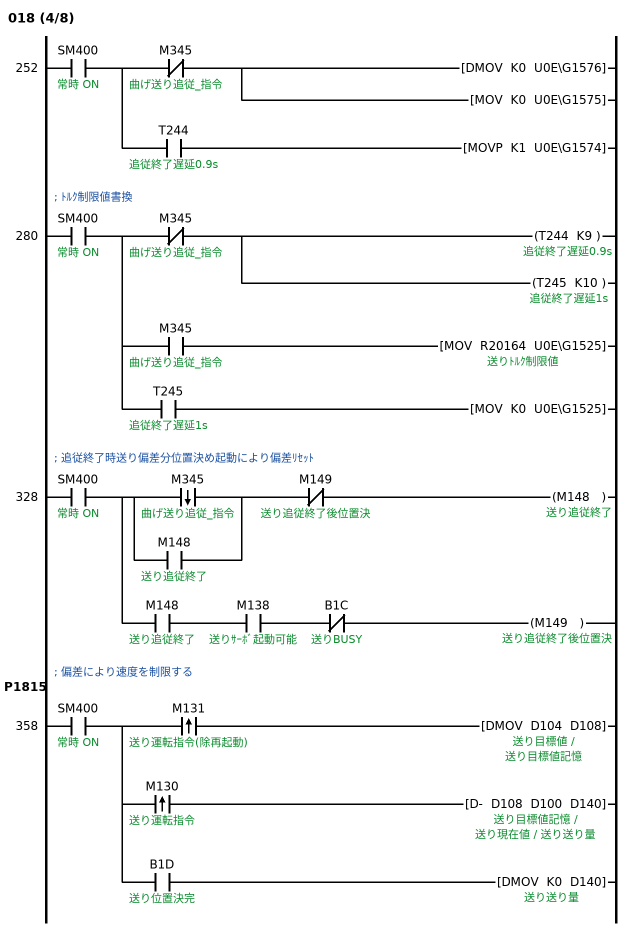
252   LD      SM400  ; 常時 ON
      MPS
      ANI     M345  ; 曲げ送り追従_指令
      DMOV    K0 U0E\G1576
      MOV     K0 U0E\G1575
      MPP
      AND     T244  ; 追従終了遅延0.9s
      MOVP    K1 U0E\G1574
; ﾄﾙｸ制限値書換
280   LD      SM400  ; 常時 ON
      MPS
      ANI     M345  ; 曲げ送り追従_指令
      OUT     T244 K9  ; 追従終了遅延0.9s
      OUT     T245 K10  ; 追従終了遅延1s
      MRD
      AND     M345  ; 曲げ送り追従_指令
      MOV     R20164 U0E\G1525  ; 送りﾄﾙｸ制限値
      MPP
      AND     T245  ; 追従終了遅延1s
      MOV     K0 U0E\G1525
; 追従終了時送り偏差分位置決め起動により偏差ﾘｾｯﾄ
328   LD      SM400  ; 常時 ON
      MPS
      LDF     M345  ; 曲げ送り追従_指令
      OR      M148  ; 送り追従終了
      ANB
      ANI     M149  ; 送り追従終了後位置決
      OUT     M148  ; 送り追従終了
      MPP
      AND     M148  ; 送り追従終了
      AND     M138  ; 送りｻｰﾎﾞ起動可能
      ANI     B1C  ; 送りBUSY
      OUT     M149  ; 送り追従終了後位置決
; 偏差により速度を制限する
; 
      P1815
358   LD      SM400  ; 常時 ON
      MPS
      ANDP    M131  ; 送り運転指令(除再起動)
      DMOV    D104 D108  ; 送り目標値記憶
      MRD
      ANDP    M130  ; 送り運転指令
      D-      D108 D100 D140  ; 送り送り量
      MPP
      AND     B1D  ; 送り位置決完
      DMOV    K0 D140
; 
      P1816
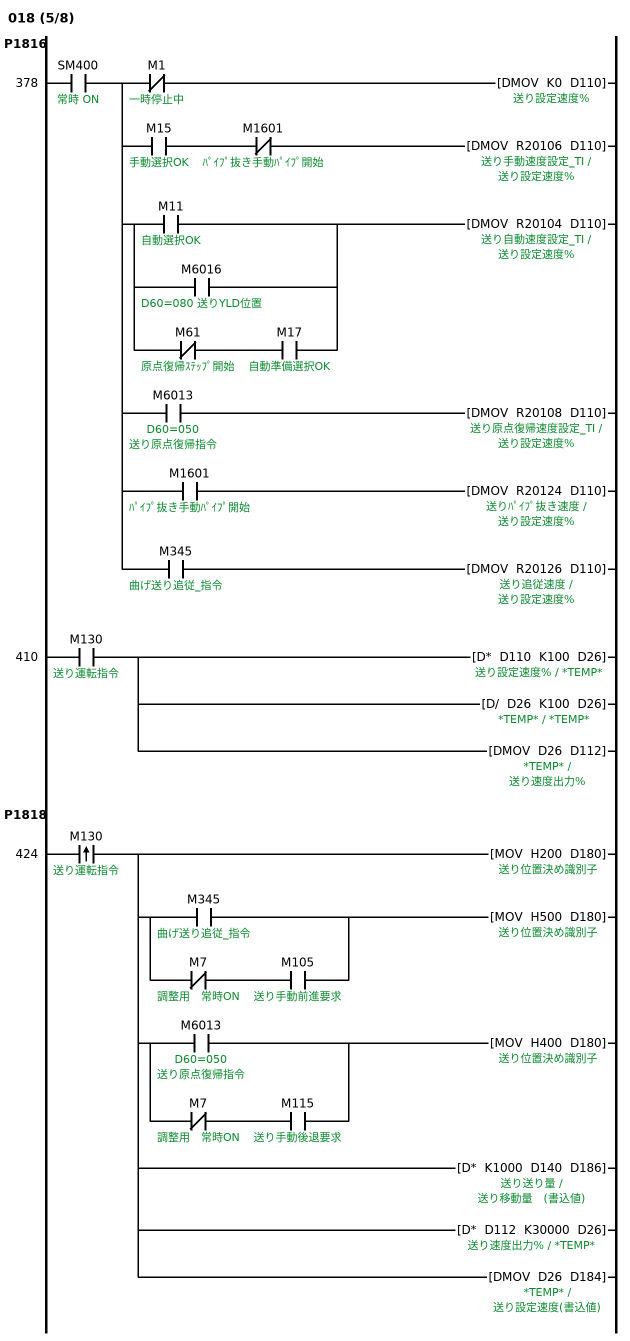
378   LD      SM400  ; 常時 ON
      MPS
      ANI     M1  ; 一時停止中
      DMOV    K0 D110  ; 送り設定速度%
      MRD
      AND     M15  ; 手動選択OK
      ANI     M1601  ; ﾊﾟｲﾌﾟ抜き手動ﾊﾟｲﾌﾟ開始
      DMOV    R20106 D110  ; 送り手動速度設定_TI
      MRD
      LD      M11  ; 自動選択OK
      OR      M6016  ; D60=080 送りYLD位置
      LDI     M61  ; 原点復帰ｽﾃｯﾌﾟ開始
      AND     M17  ; 自動準備選択OK
      ORB
      ANB
      DMOV    R20104 D110  ; 送り自動速度設定_TI
      MRD
      AND     M6013  ; D60=050 送り原点復帰指令
      DMOV    R20108 D110  ; 送り原点復帰速度設定_TI
      MRD
      AND     M1601  ; ﾊﾟｲﾌﾟ抜き手動ﾊﾟｲﾌﾟ開始
      DMOV    R20124 D110  ; 送りﾊﾟｲﾌﾟ抜き速度
      MPP
      AND     M345  ; 曲げ送り追従_指令
      DMOV    R20126 D110
410   LD      M130  ; 送り運転指令
      D*      D110 K100 D26  ; *TEMP*
      D/      D26 K100 D26
      DMOV    D26 D112  ; 送り速度出力%
; 
      P1818
424   LDP     M130  ; 送り運転指令
      MOV     H200 D180  ; 送り位置決め識別子
      MPS
      LD      M345  ; 曲げ送り追従_指令
      LDI     M7  ; 調整用　常時ON
      AND     M105  ; 送り手動前進要求
      ORB
      ANB
      MOV     H500 D180
      MRD
      LD      M6013  ; D60=050 送り原点復帰指令
      LDI     M7  ; 調整用　常時ON
      AND     M115  ; 送り手動後退要求
      ORB
      ANB
      MOV     H400 D180
      MPP
      D*      K1000 D140 D186  ; 送り移動量　(書込値)
      D*      D112 K30000 D26
      DMOV    D26 D184  ; 送り設定速度(書込値)
; 
      P1819
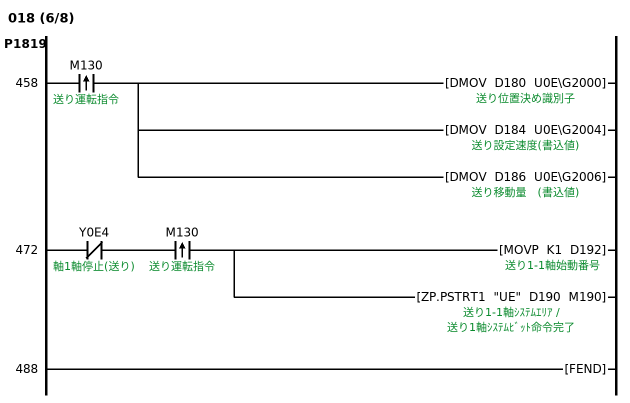
458   LDP     M130  ; 送り運転指令
      DMOV    D180 U0E\G2000
      DMOV    D184 U0E\G2004
      DMOV    D186 U0E\G2006
472   LDI     Y0E4  ; 軸1軸停止(送り)
      ANDP    M130  ; 送り運転指令
      MOVP    K1 D192  ; 送り1-1軸始動番号
      ZP.PSTRT1 "UE" D190 M190  ; 送り1-1軸ｼｽﾃﾑｴﾘｱ / 送り1軸ｼｽﾃﾑﾋﾞｯﾄ命令完了
488   FEND
; 
      P1830
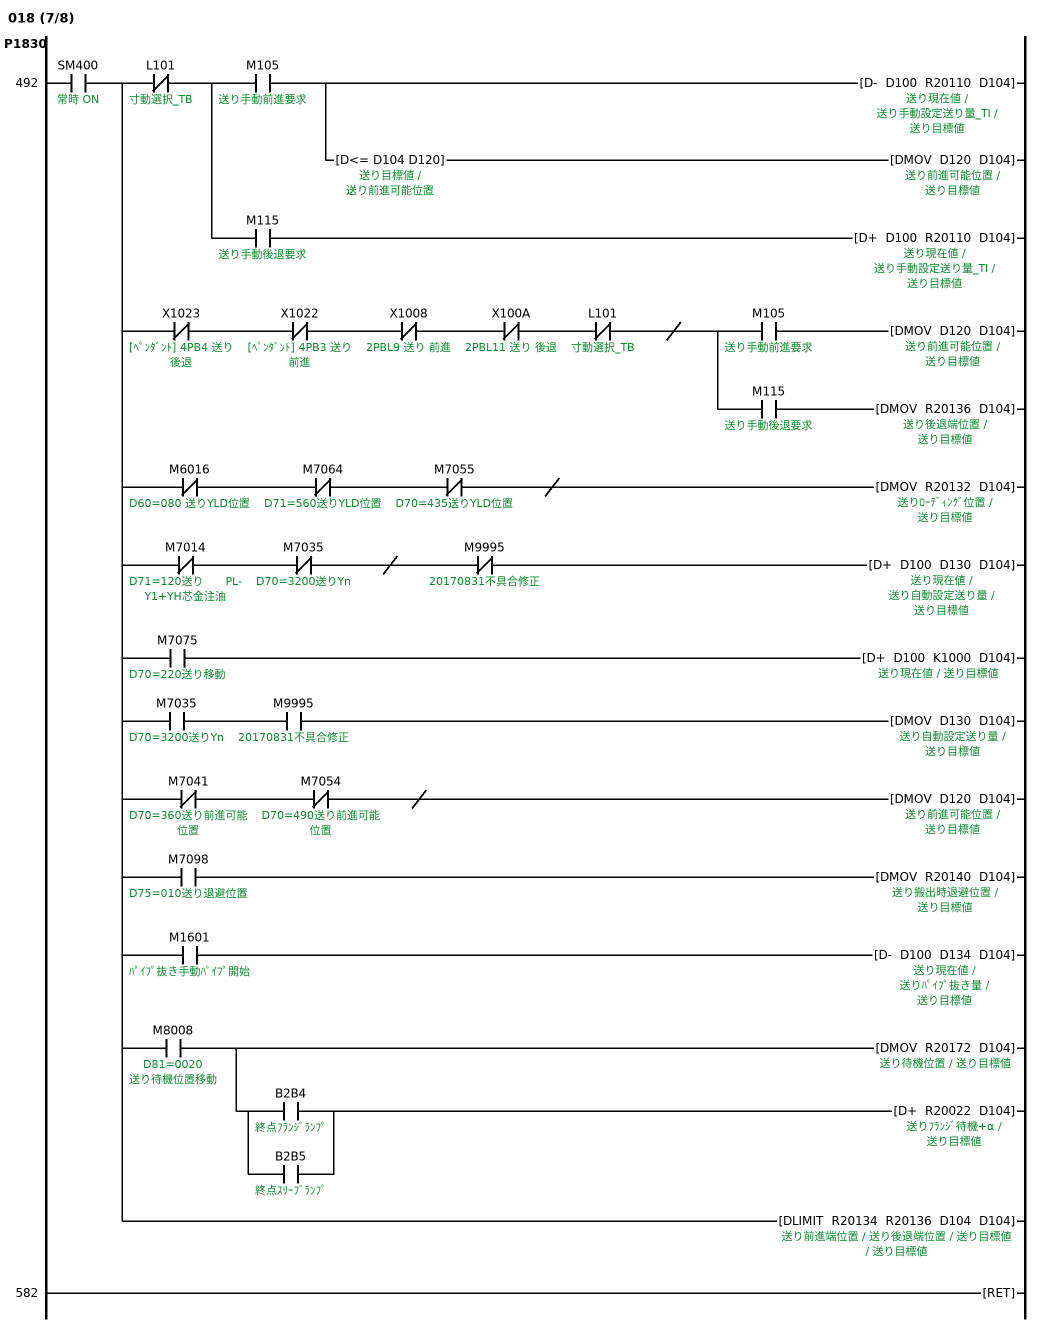
492   LD      SM400  ; 常時 ON
      MPS
      ANI     L101  ; 寸動選択_TB
      MPS
      AND     M105  ; 送り手動前進要求
      D-      D100 R20110 D104  ; 送り手動設定送り量_TI
      ANDD<=  D104 D120  ; 送り目標値 / 送り前進可能位置
      DMOV    D120 D104
      MPP
      AND     M115  ; 送り手動後退要求
      D+      D100 R20110 D104
      MRD
      ANI     X1023  ; [ﾍﾟﾝﾀﾞﾝﾄ] 4PB4 送り 後退
      ANI     X1022  ; [ﾍﾟﾝﾀﾞﾝﾄ] 4PB3 送り 前進
      ANI     X1008  ; 2PBL9 送り 前進
      ANI     X100A  ; 2PBL11 送り 後退
      ANI     L101  ; 寸動選択_TB
      INV
      MPS
      AND     M105  ; 送り手動前進要求
      DMOV    D120 D104
      MPP
      AND     M115  ; 送り手動後退要求
      DMOV    R20136 D104  ; 送り後退端位置
      MRD
      ANI     M6016  ; D60=080 送りYLD位置
      ANI     M7064  ; D71=560送りYLD位置
      ANI     M7055  ; D70=435送りYLD位置
      INV
      DMOV    R20132 D104  ; 送りﾛｰﾃﾞｨﾝｸﾞ位置
      MRD
      ANI     M7014  ; D71=120送り　　PL-Y1+YH芯金注油
      ANI     M7035  ; D70=3200送りYn
      INV
      ANI     M9995  ; 20170831不具合修正
      D+      D100 D130 D104  ; 送り自動設定送り量
      MRD
      AND     M7075  ; D70=220送り移動
      D+      D100 K1000 D104
      MRD
      AND     M7035  ; D70=3200送りYn
      AND     M9995  ; 20170831不具合修正
      DMOV    D130 D104
      MRD
      ANI     M7041  ; D70=360送り前進可能位置
      ANI     M7054  ; D70=490送り前進可能位置
      INV
      DMOV    D120 D104
      MRD
      AND     M7098  ; D75=010送り退避位置
      DMOV    R20140 D104  ; 送り搬出時退避位置
      MRD
      AND     M1601  ; ﾊﾟｲﾌﾟ抜き手動ﾊﾟｲﾌﾟ開始
      D-      D100 D134 D104  ; 送りﾊﾟｲﾌﾟ抜き量
      MRD
      AND     M8008  ; D81=0020 送り待機位置移動
      DMOV    R20172 D104  ; 送り待機位置
      LD      B2B4  ; 終点ﾌﾗﾝｼﾞﾗﾝﾌﾟ
      OR      B2B5  ; 終点ｽﾘｰﾌﾞﾗﾝﾌﾟ
      ANB
      D+      R20022 D104  ; 送りﾌﾗﾝｼﾞ待機+α
      MPP
      DLIMIT  R20134 R20136 D104 D104  ; 送り前進端位置
582   RET
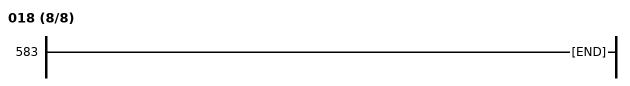
583   END
END_PROGRAM

PROGRAM 019  // 位置決めﾕﾆｯﾄ設定
; 
      P1900
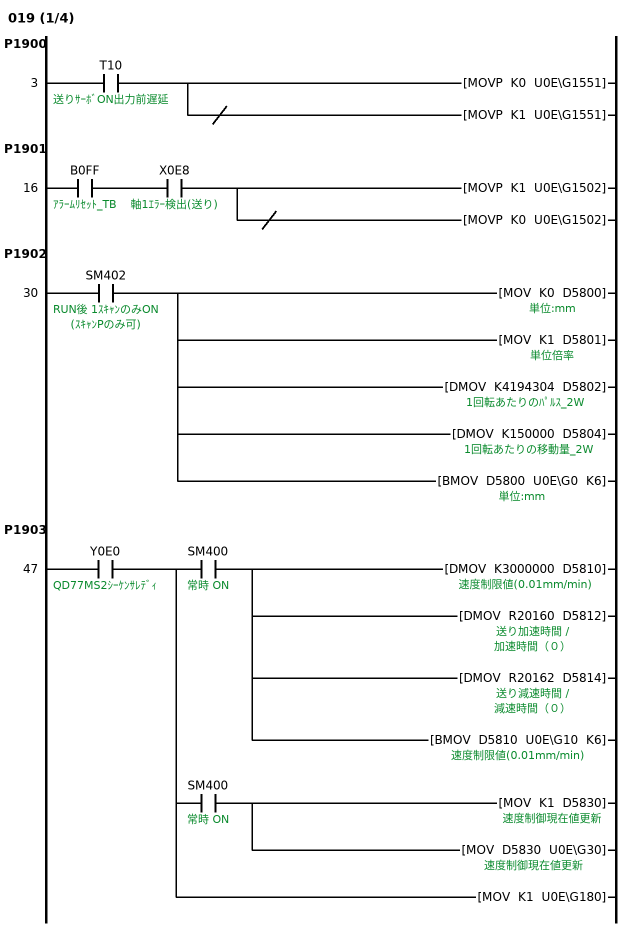
3     LD      T10  ; 送りｻｰﾎﾞON出力前遅延
      MOVP    K0 U0E\G1551
      INV
      MOVP    K1 U0E\G1551
      P1901
16    LD      B0FF  ; ｱﾗｰﾑﾘｾｯﾄ_TB
      AND     X0E8  ; 軸1ｴﾗｰ検出(送り)
      MOVP    K1 U0E\G1502
      INV
      MOVP    K0 U0E\G1502
      P1902
30    LD      SM402  ; RUN後 1ｽｷｬﾝのみON (ｽｷｬﾝPのみ可)
      MOV     K0 D5800  ; 単位:mm
      MOV     K1 D5801  ; 単位倍率
      DMOV    K4194304 D5802  ; 1回転あたりのﾊﾟﾙｽ_2W
      DMOV    K150000 D5804  ; 1回転あたりの移動量_2W
      BMOV    D5800 U0E\G0 K6
      P1903
47    LD      Y0E0  ; QD77MS2ｼｰｹﾝｻﾚﾃﾞｨ
      MPS
      AND     SM400  ; 常時 ON
      DMOV    K3000000 D5810  ; 速度制限値(0.01mm/min)
      DMOV    R20160 D5812  ; 送り加速時間 / 加速時間（０）
      DMOV    R20162 D5814  ; 送り減速時間 / 減速時間（０）
      BMOV    D5810 U0E\G10 K6
      MRD
      AND     SM400  ; 常時 ON
      MOV     K1 D5830  ; 速度制御現在値更新
      MOV     D5830 U0E\G30
      MPP
      MOV     K1 U0E\G180
      P1904
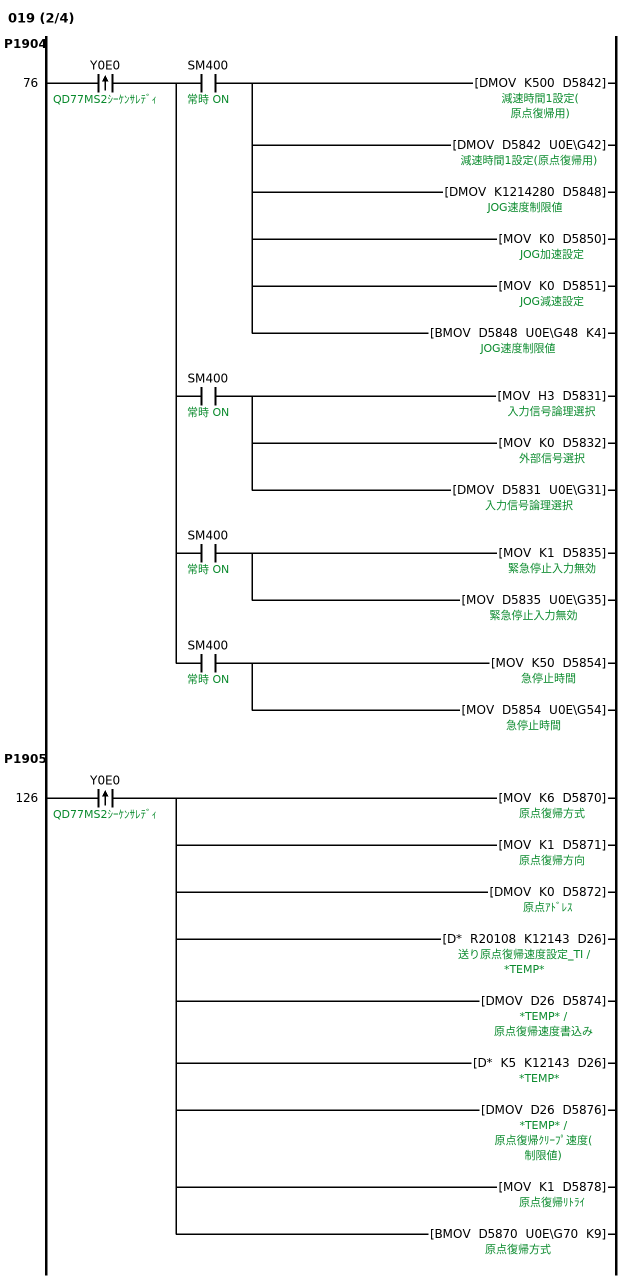
76    LDP     Y0E0  ; QD77MS2ｼｰｹﾝｻﾚﾃﾞｨ
      MPS
      AND     SM400  ; 常時 ON
      DMOV    K500 D5842  ; 減速時間1設定(原点復帰用)
      DMOV    D5842 U0E\G42
      DMOV    K1214280 D5848  ; JOG速度制限値
      MOV     K0 D5850  ; JOG加速設定
      MOV     K0 D5851  ; JOG減速設定
      BMOV    D5848 U0E\G48 K4
      MRD
      AND     SM400  ; 常時 ON
      MOV     H3 D5831  ; 入力信号論理選択
      MOV     K0 D5832  ; 外部信号選択
      DMOV    D5831 U0E\G31
      MRD
      AND     SM400  ; 常時 ON
      MOV     K1 D5835  ; 緊急停止入力無効
      MOV     D5835 U0E\G35
      MPP
      AND     SM400  ; 常時 ON
      MOV     K50 D5854  ; 急停止時間
      MOV     D5854 U0E\G54
      P1905
126   LDP     Y0E0  ; QD77MS2ｼｰｹﾝｻﾚﾃﾞｨ
      MOV     K6 D5870  ; 原点復帰方式
      MOV     K1 D5871  ; 原点復帰方向
      DMOV    K0 D5872  ; 原点ｱﾄﾞﾚｽ
      D*      R20108 K12143 D26  ; 送り原点復帰速度設定_TI / *TEMP*
      DMOV    D26 D5874  ; 原点復帰速度書込み
      D*      K5 K12143 D26
      DMOV    D26 D5876  ; 原点復帰ｸﾘｰﾌﾟ速度(制限値)
      MOV     K1 D5878  ; 原点復帰ﾘﾄﾗｲ
      BMOV    D5870 U0E\G70 K9
      P1906
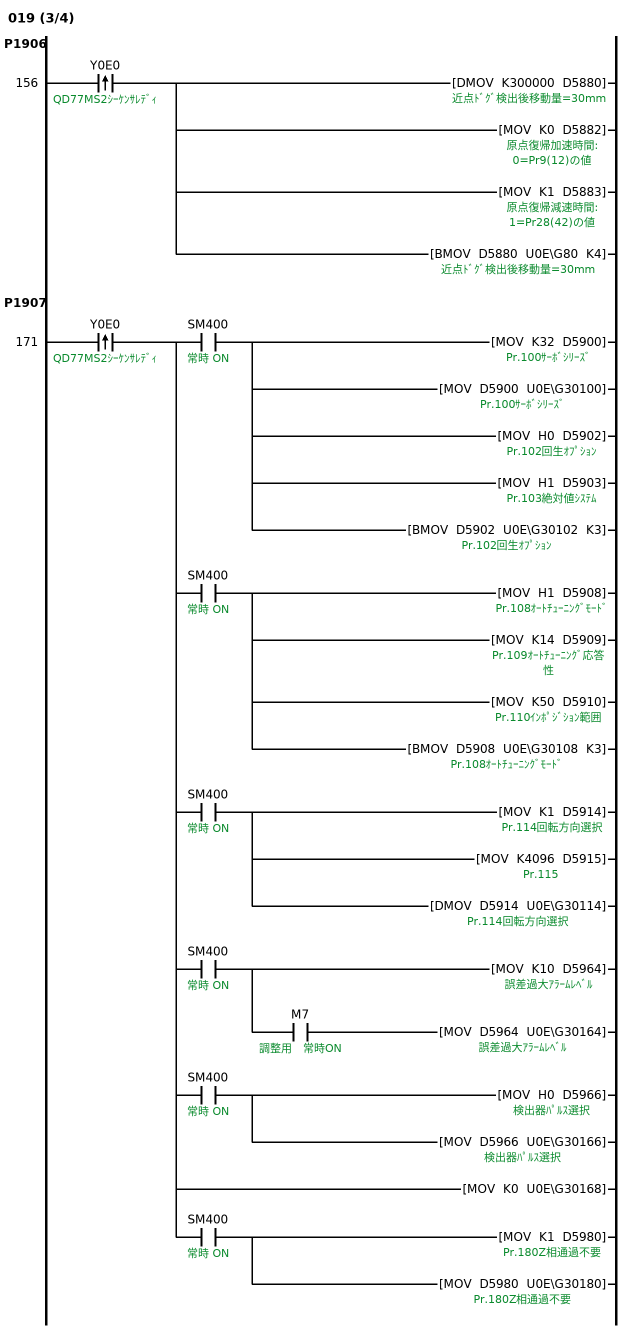
156   LDP     Y0E0  ; QD77MS2ｼｰｹﾝｻﾚﾃﾞｨ
      DMOV    K300000 D5880  ; 近点ﾄﾞｸﾞ検出後移動量=30mm
      MOV     K0 D5882  ; 原点復帰加速時間:0=Pr9(12)の値
      MOV     K1 D5883  ; 原点復帰減速時間:1=Pr28(42)の値
      BMOV    D5880 U0E\G80 K4
      P1907
171   LDP     Y0E0  ; QD77MS2ｼｰｹﾝｻﾚﾃﾞｨ
      MPS
      AND     SM400  ; 常時 ON
      MOV     K32 D5900  ; Pr.100ｻｰﾎﾞｼﾘｰｽﾞ
      MOV     D5900 U0E\G30100
      MOV     H0 D5902  ; Pr.102回生ｵﾌﾟｼｮﾝ
      MOV     H1 D5903  ; Pr.103絶対値ｼｽﾃﾑ
      BMOV    D5902 U0E\G30102 K3
      MRD
      AND     SM400  ; 常時 ON
      MOV     H1 D5908  ; Pr.108ｵｰﾄﾁｭｰﾆﾝｸﾞﾓｰﾄﾞ
      MOV     K14 D5909  ; Pr.109ｵｰﾄﾁｭｰﾆﾝｸﾞ応答性
      MOV     K50 D5910  ; Pr.110ｲﾝﾎﾟｼﾞｼｮﾝ範囲
      BMOV    D5908 U0E\G30108 K3
      MRD
      AND     SM400  ; 常時 ON
      MOV     K1 D5914  ; Pr.114回転方向選択
      MOV     K4096 D5915  ; Pr.115
      DMOV    D5914 U0E\G30114
      MRD
      AND     SM400  ; 常時 ON
      MOV     K10 D5964  ; 誤差過大ｱﾗｰﾑﾚﾍﾞﾙ
      AND     M7  ; 調整用　常時ON
      MOV     D5964 U0E\G30164
      MRD
      AND     SM400  ; 常時 ON
      MOV     H0 D5966  ; 検出器ﾊﾟﾙｽ選択
      MOV     D5966 U0E\G30166
      MPP
      MOV     K0 U0E\G30168
      AND     SM400  ; 常時 ON
      MOV     K1 D5980  ; Pr.180Z相通過不要
      MOV     D5980 U0E\G30180
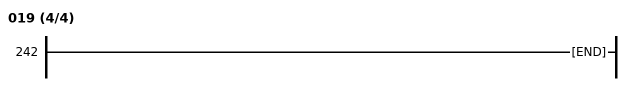
242   END
END_PROGRAM

PROGRAM 022  // ﾜｰｸﾃﾞｰﾀ読出し、書込み
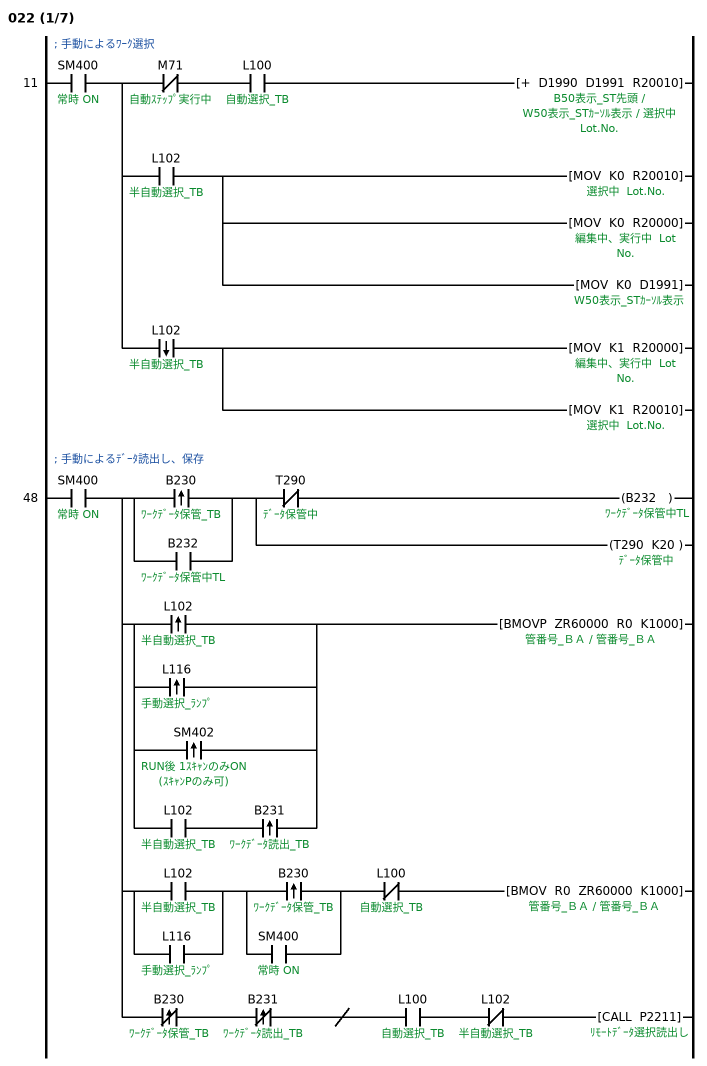
; 手動によるﾜｰｸ選択
11    LD      SM400  ; 常時 ON
      MPS
      ANI     M71  ; 自動ｽﾃｯﾌﾟ実行中
      AND     L100  ; 自動選択_TB
      +       D1990 D1991 R20010  ; B50表示_ST先頭 / W50表示_STｶｰｿﾙ表示 / 選択中  Lot.No.
      MRD
      AND     L102  ; 半自動選択_TB
      MOV     K0 R20010
      MOV     K0 R20000  ; 編集中、実行中  Lot No.
      MOV     K0 D1991
      MPP
      ANDF    L102  ; 半自動選択_TB
      MOV     K1 R20000
      MOV     K1 R20010
; 手動によるﾃﾞｰﾀ読出し、保存
48    LD      SM400  ; 常時 ON
      MPS
      LDP     B230  ; ﾜｰｸﾃﾞｰﾀ保管_TB
      OR      B232  ; ﾜｰｸﾃﾞｰﾀ保管中TL
      ANB
      MPS
      ANI     T290  ; ﾃﾞｰﾀ保管中
      OUT     B232  ; ﾜｰｸﾃﾞｰﾀ保管中TL
      MPP
      OUT     T290 K20  ; ﾃﾞｰﾀ保管中
      MRD
      LDP     L102  ; 半自動選択_TB
      ORP     L116  ; 手動選択_ﾗﾝﾌﾟ
      ORP     SM402  ; RUN後 1ｽｷｬﾝのみON (ｽｷｬﾝPのみ可)
      LD      L102  ; 半自動選択_TB
      ANDP    B231  ; ﾜｰｸﾃﾞｰﾀ読出_TB
      ORB
      ANB
      BMOVP   ZR60000 R0 K1000  ; 管番号_ＢＡ / 管番号_ＢＡ
      MRD
      LD      L102  ; 半自動選択_TB
      OR      L116  ; 手動選択_ﾗﾝﾌﾟ
      ANB
      LDP     B230  ; ﾜｰｸﾃﾞｰﾀ保管_TB
      OR      SM400  ; 常時 ON
      ANB
      ANI     L100  ; 自動選択_TB
      BMOV    R0 ZR60000 K1000
      MPP
      ANDPI   B230  ; ﾜｰｸﾃﾞｰﾀ保管_TB
      ANDPI   B231  ; ﾜｰｸﾃﾞｰﾀ読出_TB
      INV
      AND     L100  ; 自動選択_TB
      ANI     L102  ; 半自動選択_TB
      CALL    P2211  ; ﾘﾓｰﾄﾃﾞｰﾀ選択読出し
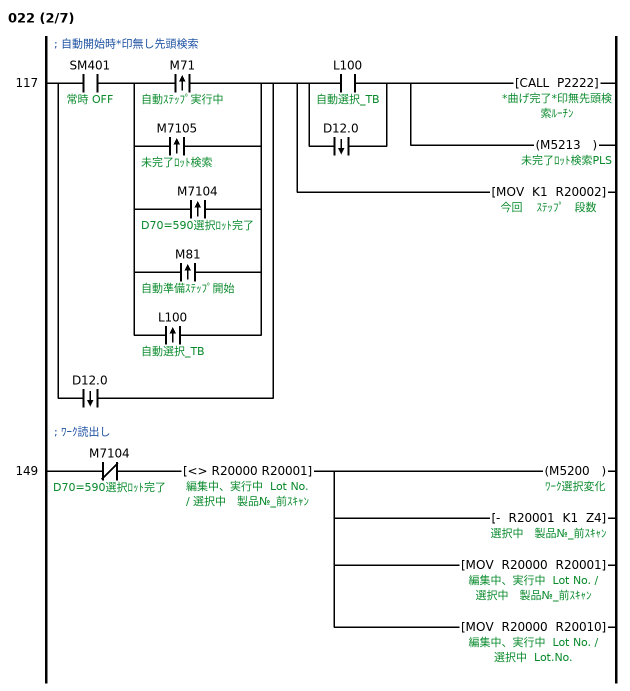
; 自動開始時*印無し先頭検索
117   LD      SM401  ; 常時 OFF
      LDP     M71  ; 自動ｽﾃｯﾌﾟ実行中
      ORP     M7105  ; 未完了ﾛｯﾄ検索
      ORP     M7104  ; D70=590選択ﾛｯﾄ完了
      ORP     M81  ; 自動準備ｽﾃｯﾌﾟ開始
      ORP     L100  ; 自動選択_TB
      ANB
      ORF     D12.0
      MPS
      LD      L100  ; 自動選択_TB
      ORF     D12.0
      ANB
      CALL    P2222  ; *曲げ完了*印無先頭検索ﾙｰﾁﾝ
      OUT     M5213  ; 未完了ﾛｯﾄ検索PLS
      MPP
      MOV     K1 R20002  ; 今回    ｽﾃｯﾌﾟ   段数
; ﾜｰｸ読出し
149   LDI     M7104  ; D70=590選択ﾛｯﾄ完了
      AND<>   R20000 R20001  ; 編集中、実行中  Lot No. / 選択中　製品№_前ｽｷｬﾝ
      OUT     M5200  ; ﾜｰｸ選択変化
      -       R20001 K1 Z4
      MOV     R20000 R20001
      MOV     R20000 R20010
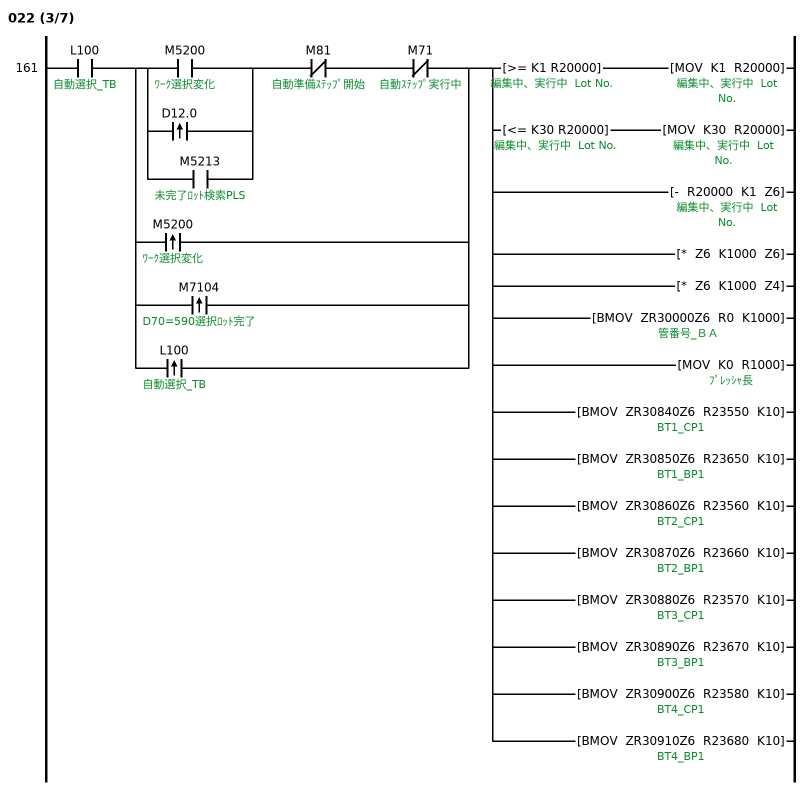
161   LD      L100  ; 自動選択_TB
      LD      M5200  ; ﾜｰｸ選択変化
      ORP     D12.0
      OR      M5213  ; 未完了ﾛｯﾄ検索PLS
      ANI     M81  ; 自動準備ｽﾃｯﾌﾟ開始
      ANI     M71  ; 自動ｽﾃｯﾌﾟ実行中
      ORP     M5200  ; ﾜｰｸ選択変化
      ORP     M7104  ; D70=590選択ﾛｯﾄ完了
      ORP     L100  ; 自動選択_TB
      ANB
      MPS
      AND>=   K1 R20000  ; 編集中、実行中  Lot No.
      MOV     K1 R20000
      MRD
      AND<=   K30 R20000  ; 編集中、実行中  Lot No.
      MOV     K30 R20000
      MPP
      -       R20000 K1 Z6
      *       Z6 K1000 Z6
      *       Z6 K1000 Z4
      BMOV    ZR30000Z6 R0 K1000
      MOV     K0 R1000  ; ﾌﾟﾚｯｼｬ長
      BMOV    ZR30840Z6 R23550 K10  ; BT1_CP1
      BMOV    ZR30850Z6 R23650 K10  ; BT1_BP1
      BMOV    ZR30860Z6 R23560 K10  ; BT2_CP1
      BMOV    ZR30870Z6 R23660 K10  ; BT2_BP1
      BMOV    ZR30880Z6 R23570 K10  ; BT3_CP1
      BMOV    ZR30890Z6 R23670 K10  ; BT3_BP1
      BMOV    ZR30900Z6 R23580 K10  ; BT4_CP1
      BMOV    ZR30910Z6 R23680 K10  ; BT4_BP1
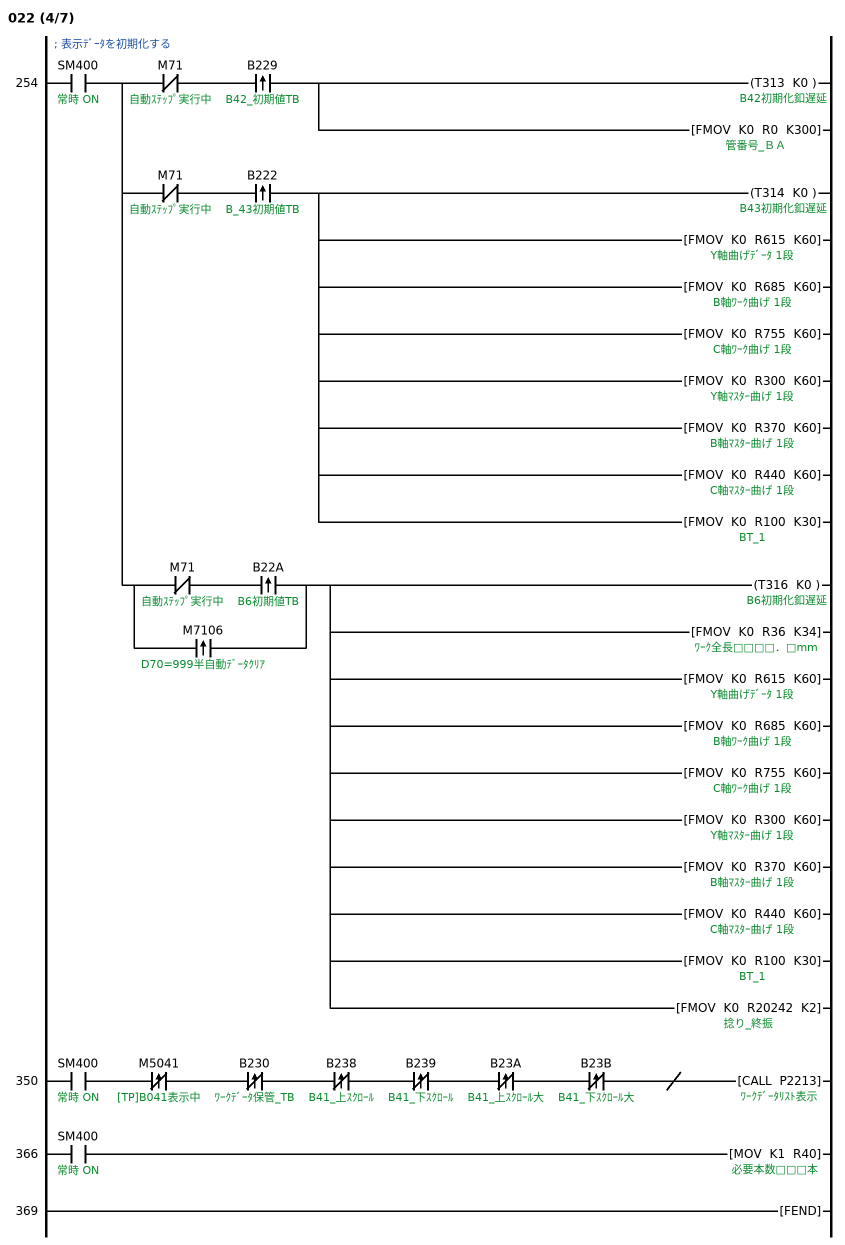
; 表示ﾃﾞｰﾀを初期化する
254   LD      SM400  ; 常時 ON
      MPS
      ANI     M71  ; 自動ｽﾃｯﾌﾟ実行中
      ANDP    B229  ; B42_初期値TB
      OUT     T313 K0  ; B42初期化釦遅延
      FMOV    K0 R0 K300
      MRD
      ANI     M71  ; 自動ｽﾃｯﾌﾟ実行中
      ANDP    B222  ; B_43初期値TB
      OUT     T314 K0  ; B43初期化釦遅延
      FMOV    K0 R615 K60  ; Y軸曲げﾃﾞｰﾀ 1段
      FMOV    K0 R685 K60  ; B軸ﾜｰｸ曲げ 1段
      FMOV    K0 R755 K60  ; C軸ﾜｰｸ曲げ 1段
      FMOV    K0 R300 K60  ; Y軸ﾏｽﾀｰ曲げ 1段
      FMOV    K0 R370 K60  ; B軸ﾏｽﾀｰ曲げ 1段
      FMOV    K0 R440 K60  ; C軸ﾏｽﾀｰ曲げ 1段
      FMOV    K0 R100 K30  ; BT_1
      MPP
      LDI     M71  ; 自動ｽﾃｯﾌﾟ実行中
      ANDP    B22A  ; B6初期値TB
      ORP     M7106  ; D70=999半自動ﾃﾞｰﾀｸﾘｱ
      ANB
      OUT     T316 K0  ; B6初期化釦遅延
      FMOV    K0 R36 K34  ; ﾜｰｸ全長□□□□．□mm
      FMOV    K0 R615 K60
      FMOV    K0 R685 K60
      FMOV    K0 R755 K60
      FMOV    K0 R300 K60
      FMOV    K0 R370 K60
      FMOV    K0 R440 K60
      FMOV    K0 R100 K30
      FMOV    K0 R20242 K2  ; 捻り_終振
350   LD      SM400  ; 常時 ON
      ANDPI   M5041  ; [TP]B041表示中
      ANDPI   B230  ; ﾜｰｸﾃﾞｰﾀ保管_TB
      ANDPI   B238  ; B41_上ｽｸﾛｰﾙ
      ANDPI   B239  ; B41_下ｽｸﾛｰﾙ
      ANDPI   B23A  ; B41_上ｽｸﾛｰﾙ大
      ANDPI   B23B  ; B41_下ｽｸﾛｰﾙ大
      INV
      CALL    P2213  ; ﾜｰｸﾃﾞｰﾀﾘｽﾄ表示
366   LD      SM400  ; 常時 ON
      MOV     K1 R40  ; 必要本数□□□本
369   FEND
; ﾘﾓｰﾄﾃﾞｰﾀのｽｲｯﾁによるﾃﾞｰﾀ読出し、書込み
      P2211
